(* Logix 5000 project; controller reports 1756-L63 rev 20.15; software revision 20.04; part 8 of 52 *)

        [734].log_data[9].valid := 1, [734].log_data[10].valid := 1, [734].log_data[11].valid := 1, [734].log_data[12].valid := 1, [734].log_data[13].valid := 1, [734].log_data[14].valid := 1, [734].log_data[15].valid := 1, [734].log_data[16].valid := 1, [734].log_data[17].valid := 1, [734].log_data[18].valid := 1, [734].log_data[19].valid := 1, [734].time.Year := 2023, [734].time.Month := 1, [734].time.Day := 15, [734].time.Hour := 7, [734].time.Minute := 59, [734].time.Second := 59, [735].log_data[0].min := 1.0, [735].log_data[0].max := 1.0, [735].log_data[0].total := 900.0, [735].log_data[0].time := 900.0, [735].log_data[0].valid := 1, [735].log_data[1].valid := 1, [735].log_data[2].valid := 1, [735].log_data[3].valid := 1, [735].log_data[4].valid := 1, [735].log_data[5].valid := 1, [735].log_data[6].valid := 1, [735].log_data[7].valid := 1, [735].log_data[8].valid := 1, [735].log_data[9].valid := 1, [735].log_data[10].valid := 1, [735].log_data[11].valid := 1, [735].log_data[12].valid := 1, [735].log_data[13].valid := 1, [735].log_data[14].valid := 1, [735].log_data[15].valid := 1, [735].log_data[16].valid := 1, [735].log_data[17].valid := 1, [735].log_data[18].valid := 1, [735].log_data[19].valid := 1, [735].time.Year := 2023, [735].time.Month := 1, [735].time.Day := 15, [735].time.Hour := 8, [735].time.Minute := 14, [735].time.Second := 59, [736].log_data[0].min := 1.0, [736].log_data[0].max := 1.0, [736].log_data[0].total := 900.0, [736].log_data[0].time := 900.0, [736].log_data[0].minminute := 15, [736].log_data[0].maxminute := 15, [736].log_data[0].valid := 1, [736].log_data[1].valid := 1, [736].log_data[2].valid := 1, [736].log_data[3].valid := 1, [736].log_data[4].valid := 1, [736].log_data[5].valid := 1, [736].log_data[6].valid := 1,
        [736].log_data[7].valid := 1, [736].log_data[8].valid := 1, [736].log_data[9].valid := 1, [736].log_data[10].valid := 1, [736].log_data[11].valid := 1, [736].log_data[12].valid := 1, [736].log_data[13].valid := 1, [736].log_data[14].valid := 1, [736].log_data[15].valid := 1, [736].log_data[16].valid := 1, [736].log_data[17].valid := 1, [736].log_data[18].valid := 1, [736].log_data[19].valid := 1, [736].time.Year := 2023, [736].time.Month := 1, [736].time.Day := 15, [736].time.Hour := 8, [736].time.Minute := 29, [736].time.Second := 59, [737].log_data[0].min := 1.0, [737].log_data[0].max := 1.0, [737].log_data[0].total := 900.0, [737].log_data[0].time := 900.0, [737].log_data[0].minminute := 30, [737].log_data[0].maxminute := 30, [737].log_data[0].valid := 1, [737].log_data[1].valid := 1, [737].log_data[2].valid := 1, [737].log_data[3].valid := 1, [737].log_data[4].valid := 1, [737].log_data[5].valid := 1, [737].log_data[6].valid := 1, [737].log_data[7].valid := 1, [737].log_data[8].valid := 1, [737].log_data[9].valid := 1, [737].log_data[10].valid := 1, [737].log_data[11].valid := 1, [737].log_data[12].valid := 1, [737].log_data[13].valid := 1, [737].log_data[14].valid := 1, [737].log_data[15].valid := 1, [737].log_data[16].valid := 1, [737].log_data[17].valid := 1, [737].log_data[18].valid := 1, [737].log_data[19].valid := 1, [737].time.Year := 2023, [737].time.Month := 1, [737].time.Day := 15, [737].time.Hour := 8, [737].time.Minute := 44, [737].time.Second := 59, [738].log_data[0].min := 1.0, [738].log_data[0].max := 1.0, [738].log_data[0].total := 900.0, [738].log_data[0].time := 900.0, [738].log_data[0].minminute := 45, [738].log_data[0].maxminute := 45, [738].log_data[0].valid := 1, [738].log_data[1].valid := 1, [738].log_data[2].valid := 1,
        [738].log_data[3].valid := 1, [738].log_data[4].valid := 1, [738].log_data[5].valid := 1, [738].log_data[6].valid := 1, [738].log_data[7].valid := 1, [738].log_data[8].valid := 1, [738].log_data[9].valid := 1, [738].log_data[10].valid := 1, [738].log_data[11].valid := 1, [738].log_data[12].valid := 1, [738].log_data[13].valid := 1, [738].log_data[14].valid := 1, [738].log_data[15].valid := 1, [738].log_data[16].valid := 1, [738].log_data[17].valid := 1, [738].log_data[18].valid := 1, [738].log_data[19].valid := 1, [738].time.Year := 2023, [738].time.Month := 1, [738].time.Day := 15, [738].time.Hour := 8, [738].time.Minute := 59, [738].time.Second := 59, [739].log_data[0].min := 1.0, [739].log_data[0].max := 1.0, [739].log_data[0].total := 900.0, [739].log_data[0].time := 900.0, [739].log_data[0].valid := 1, [739].log_data[1].valid := 1, [739].log_data[2].valid := 1, [739].log_data[3].valid := 1, [739].log_data[4].valid := 1, [739].log_data[5].valid := 1, [739].log_data[6].valid := 1, [739].log_data[7].valid := 1, [739].log_data[8].valid := 1, [739].log_data[9].valid := 1, [739].log_data[10].valid := 1, [739].log_data[11].valid := 1, [739].log_data[12].valid := 1, [739].log_data[13].valid := 1, [739].log_data[14].valid := 1, [739].log_data[15].valid := 1, [739].log_data[16].valid := 1, [739].log_data[17].valid := 1, [739].log_data[18].valid := 1, [739].log_data[19].valid := 1, [739].time.Year := 2023, [739].time.Month := 1, [739].time.Day := 15, [739].time.Hour := 9, [739].time.Minute := 14, [739].time.Second := 59, [740].log_data[0].min := 1.0, [740].log_data[0].max := 1.0, [740].log_data[0].total := 900.0, [740].log_data[0].time := 900.0, [740].log_data[0].minminute := 15, [740].log_data[0].maxminute := 15, [740].log_data[0].valid := 1,
        [740].log_data[1].valid := 1, [740].log_data[2].valid := 1, [740].log_data[3].valid := 1, [740].log_data[4].valid := 1, [740].log_data[5].valid := 1, [740].log_data[6].valid := 1, [740].log_data[7].valid := 1, [740].log_data[8].valid := 1, [740].log_data[9].valid := 1, [740].log_data[10].valid := 1, [740].log_data[11].valid := 1, [740].log_data[12].valid := 1, [740].log_data[13].valid := 1, [740].log_data[14].valid := 1, [740].log_data[15].valid := 1, [740].log_data[16].valid := 1, [740].log_data[17].valid := 1, [740].log_data[18].valid := 1, [740].log_data[19].valid := 1, [740].time.Year := 2023, [740].time.Month := 1, [740].time.Day := 15, [740].time.Hour := 9, [740].time.Minute := 29, [740].time.Second := 59, [741].log_data[0].min := 1.0, [741].log_data[0].max := 1.0, [741].log_data[0].total := 900.0, [741].log_data[0].time := 900.0, [741].log_data[0].minminute := 30, [741].log_data[0].maxminute := 30, [741].log_data[0].valid := 1, [741].log_data[1].valid := 1, [741].log_data[2].valid := 1, [741].log_data[3].valid := 1, [741].log_data[4].valid := 1, [741].log_data[5].valid := 1, [741].log_data[6].valid := 1, [741].log_data[7].valid := 1, [741].log_data[8].valid := 1, [741].log_data[9].valid := 1, [741].log_data[10].valid := 1, [741].log_data[11].valid := 1, [741].log_data[12].valid := 1, [741].log_data[13].valid := 1, [741].log_data[14].valid := 1, [741].log_data[15].valid := 1, [741].log_data[16].valid := 1, [741].log_data[17].valid := 1, [741].log_data[18].valid := 1, [741].log_data[19].valid := 1, [741].time.Year := 2023, [741].time.Month := 1, [741].time.Day := 15, [741].time.Hour := 9, [741].time.Minute := 44, [741].time.Second := 59, [742].log_data[0].min := 1.0, [742].log_data[0].max := 1.0, [742].log_data[0].total := 900.0,
        [742].log_data[0].time := 900.0, [742].log_data[0].minminute := 45, [742].log_data[0].maxminute := 45, [742].log_data[0].valid := 1, [742].log_data[1].valid := 1, [742].log_data[2].valid := 1, [742].log_data[3].valid := 1, [742].log_data[4].valid := 1, [742].log_data[5].valid := 1, [742].log_data[6].valid := 1, [742].log_data[7].valid := 1, [742].log_data[8].valid := 1, [742].log_data[9].valid := 1, [742].log_data[10].valid := 1, [742].log_data[11].valid := 1, [742].log_data[12].valid := 1, [742].log_data[13].valid := 1, [742].log_data[14].valid := 1, [742].log_data[15].valid := 1, [742].log_data[16].valid := 1, [742].log_data[17].valid := 1, [742].log_data[18].valid := 1, [742].log_data[19].valid := 1, [742].time.Year := 2023, [742].time.Month := 1, [742].time.Day := 15, [742].time.Hour := 9, [742].time.Minute := 59, [742].time.Second := 59, [743].log_data[0].min := 1.0, [743].log_data[0].max := 1.0, [743].log_data[0].total := 900.0, [743].log_data[0].time := 900.0, [743].log_data[0].valid := 1, [743].log_data[1].valid := 1, [743].log_data[2].valid := 1, [743].log_data[3].valid := 1, [743].log_data[4].valid := 1, [743].log_data[5].valid := 1, [743].log_data[6].valid := 1, [743].log_data[7].valid := 1, [743].log_data[8].valid := 1, [743].log_data[9].valid := 1, [743].log_data[10].valid := 1, [743].log_data[11].valid := 1, [743].log_data[12].valid := 1, [743].log_data[13].valid := 1, [743].log_data[14].valid := 1, [743].log_data[15].valid := 1, [743].log_data[16].valid := 1, [743].log_data[17].valid := 1, [743].log_data[18].valid := 1, [743].log_data[19].valid := 1, [743].time.Year := 2023, [743].time.Month := 1, [743].time.Day := 15, [743].time.Hour := 10, [743].time.Minute := 14, [743].time.Second := 59, [744].log_data[0].min := 1.0,
        [744].log_data[0].max := 1.0, [744].log_data[0].total := 900.0, [744].log_data[0].time := 900.0, [744].log_data[0].minminute := 15, [744].log_data[0].maxminute := 15, [744].log_data[0].valid := 1, [744].log_data[1].valid := 1, [744].log_data[2].valid := 1, [744].log_data[3].valid := 1, [744].log_data[4].valid := 1, [744].log_data[5].valid := 1, [744].log_data[6].valid := 1, [744].log_data[7].valid := 1, [744].log_data[8].valid := 1, [744].log_data[9].valid := 1, [744].log_data[10].valid := 1, [744].log_data[11].valid := 1, [744].log_data[12].valid := 1, [744].log_data[13].valid := 1, [744].log_data[14].valid := 1, [744].log_data[15].valid := 1, [744].log_data[16].valid := 1, [744].log_data[17].valid := 1, [744].log_data[18].valid := 1, [744].log_data[19].valid := 1, [744].time.Year := 2023, [744].time.Month := 1, [744].time.Day := 15, [744].time.Hour := 10, [744].time.Minute := 29, [744].time.Second := 59, [745].log_data[0].min := 1.0, [745].log_data[0].max := 1.0, [745].log_data[0].total := 900.0, [745].log_data[0].time := 900.0, [745].log_data[0].minminute := 30, [745].log_data[0].maxminute := 30, [745].log_data[0].valid := 1, [745].log_data[1].valid := 1, [745].log_data[2].valid := 1, [745].log_data[3].valid := 1, [745].log_data[4].valid := 1, [745].log_data[5].valid := 1, [745].log_data[6].valid := 1, [745].log_data[7].valid := 1, [745].log_data[8].valid := 1, [745].log_data[9].valid := 1, [745].log_data[10].valid := 1, [745].log_data[11].valid := 1, [745].log_data[12].valid := 1, [745].log_data[13].valid := 1, [745].log_data[14].valid := 1, [745].log_data[15].valid := 1, [745].log_data[16].valid := 1, [745].log_data[17].valid := 1, [745].log_data[18].valid := 1, [745].log_data[19].valid := 1, [745].time.Year := 2023, [745].time.Month := 1, [745].time.Day := 15,
        [745].time.Hour := 10, [745].time.Minute := 44, [745].time.Second := 59, [746].log_data[0].min := 1.0, [746].log_data[0].max := 1.0, [746].log_data[0].total := 900.0, [746].log_data[0].time := 900.0, [746].log_data[0].minminute := 45, [746].log_data[0].maxminute := 45, [746].log_data[0].valid := 1, [746].log_data[1].valid := 1, [746].log_data[2].valid := 1, [746].log_data[3].valid := 1, [746].log_data[4].valid := 1, [746].log_data[5].valid := 1, [746].log_data[6].valid := 1, [746].log_data[7].valid := 1, [746].log_data[8].valid := 1, [746].log_data[9].valid := 1, [746].log_data[10].valid := 1, [746].log_data[11].valid := 1, [746].log_data[12].valid := 1, [746].log_data[13].valid := 1, [746].log_data[14].valid := 1, [746].log_data[15].valid := 1, [746].log_data[16].valid := 1, [746].log_data[17].valid := 1, [746].log_data[18].valid := 1, [746].log_data[19].valid := 1, [746].time.Year := 2023, [746].time.Month := 1, [746].time.Day := 15, [746].time.Hour := 10, [746].time.Minute := 59, [746].time.Second := 59, [747].log_data[0].min := 1.0, [747].log_data[0].max := 1.0, [747].log_data[0].total := 899.5, [747].log_data[0].time := 899.5, [747].log_data[0].valid := 1, [747].log_data[1].valid := 1, [747].log_data[2].valid := 1, [747].log_data[3].valid := 1, [747].log_data[4].valid := 1, [747].log_data[5].valid := 1, [747].log_data[6].valid := 1, [747].log_data[7].valid := 1, [747].log_data[8].valid := 1, [747].log_data[9].valid := 1, [747].log_data[10].valid := 1, [747].log_data[11].valid := 1, [747].log_data[12].valid := 1, [747].log_data[13].valid := 1, [747].log_data[14].valid := 1, [747].log_data[15].valid := 1, [747].log_data[16].valid := 1, [747].log_data[17].valid := 1, [747].log_data[18].valid := 1, [747].log_data[19].valid := 1, [747].time.Year := 2023,
        [747].time.Month := 1, [747].time.Day := 15, [747].time.Hour := 11, [747].time.Minute := 14, [747].time.Second := 59, [748].log_data[0].min := 1.0, [748].log_data[0].max := 1.0, [748].log_data[0].total := 900.0, [748].log_data[0].time := 900.0, [748].log_data[0].minminute := 15, [748].log_data[0].maxminute := 15, [748].log_data[0].valid := 1, [748].log_data[1].valid := 1, [748].log_data[2].valid := 1, [748].log_data[3].valid := 1, [748].log_data[4].valid := 1, [748].log_data[5].valid := 1, [748].log_data[6].valid := 1, [748].log_data[7].valid := 1, [748].log_data[8].valid := 1, [748].log_data[9].valid := 1, [748].log_data[10].valid := 1, [748].log_data[11].valid := 1, [748].log_data[12].valid := 1, [748].log_data[13].valid := 1, [748].log_data[14].valid := 1, [748].log_data[15].valid := 1, [748].log_data[16].valid := 1, [748].log_data[17].valid := 1, [748].log_data[18].valid := 1, [748].log_data[19].valid := 1, [748].time.Year := 2023, [748].time.Month := 1, [748].time.Day := 15, [748].time.Hour := 11, [748].time.Minute := 29, [748].time.Second := 59, [749].log_data[0].min := 1.0, [749].log_data[0].max := 1.0, [749].log_data[0].total := 900.0, [749].log_data[0].time := 900.0, [749].log_data[0].minminute := 30, [749].log_data[0].maxminute := 30, [749].log_data[0].valid := 1, [749].log_data[1].valid := 1, [749].log_data[2].valid := 1, [749].log_data[3].valid := 1, [749].log_data[4].valid := 1, [749].log_data[5].valid := 1, [749].log_data[6].valid := 1, [749].log_data[7].valid := 1, [749].log_data[8].valid := 1, [749].log_data[9].valid := 1, [749].log_data[10].valid := 1, [749].log_data[11].valid := 1, [749].log_data[12].valid := 1, [749].log_data[13].valid := 1, [749].log_data[14].valid := 1, [749].log_data[15].valid := 1, [749].log_data[16].valid := 1,
        [749].log_data[17].valid := 1, [749].log_data[18].valid := 1, [749].log_data[19].valid := 1, [749].time.Year := 2023, [749].time.Month := 1, [749].time.Day := 15, [749].time.Hour := 11, [749].time.Minute := 44, [749].time.Second := 59, [750].log_data[0].min := 1.0, [750].log_data[0].max := 1.0, [750].log_data[0].total := 900.0, [750].log_data[0].time := 900.0, [750].log_data[0].minminute := 45, [750].log_data[0].maxminute := 45, [750].log_data[0].valid := 1, [750].log_data[1].valid := 1, [750].log_data[2].valid := 1, [750].log_data[3].valid := 1, [750].log_data[4].valid := 1, [750].log_data[5].valid := 1, [750].log_data[6].valid := 1, [750].log_data[7].valid := 1, [750].log_data[8].valid := 1, [750].log_data[9].valid := 1, [750].log_data[10].valid := 1, [750].log_data[11].valid := 1, [750].log_data[12].valid := 1, [750].log_data[13].valid := 1, [750].log_data[14].valid := 1, [750].log_data[15].valid := 1, [750].log_data[16].valid := 1, [750].log_data[17].valid := 1, [750].log_data[18].valid := 1, [750].log_data[19].valid := 1, [750].time.Year := 2023, [750].time.Month := 1, [750].time.Day := 15, [750].time.Hour := 11, [750].time.Minute := 59, [750].time.Second := 59, [751].log_data[0].min := 1.0, [751].log_data[0].max := 1.0, [751].log_data[0].total := 900.0, [751].log_data[0].time := 900.0, [751].log_data[0].valid := 1, [751].log_data[1].valid := 1, [751].log_data[2].valid := 1, [751].log_data[3].valid := 1, [751].log_data[4].valid := 1, [751].log_data[5].valid := 1, [751].log_data[6].valid := 1, [751].log_data[7].valid := 1, [751].log_data[8].valid := 1, [751].log_data[9].valid := 1, [751].log_data[10].valid := 1, [751].log_data[11].valid := 1, [751].log_data[12].valid := 1, [751].log_data[13].valid := 1, [751].log_data[14].valid := 1,
        [751].log_data[15].valid := 1, [751].log_data[16].valid := 1, [751].log_data[17].valid := 1, [751].log_data[18].valid := 1, [751].log_data[19].valid := 1, [751].time.Year := 2023, [751].time.Month := 1, [751].time.Day := 15, [751].time.Hour := 12, [751].time.Minute := 14, [751].time.Second := 59, [752].log_data[0].min := 1.0, [752].log_data[0].max := 1.0, [752].log_data[0].total := 900.0, [752].log_data[0].time := 900.0, [752].log_data[0].minminute := 15, [752].log_data[0].maxminute := 15, [752].log_data[0].valid := 1, [752].log_data[1].valid := 1, [752].log_data[2].valid := 1, [752].log_data[3].valid := 1, [752].log_data[4].valid := 1, [752].log_data[5].valid := 1, [752].log_data[6].valid := 1, [752].log_data[7].valid := 1, [752].log_data[8].valid := 1, [752].log_data[9].valid := 1, [752].log_data[10].valid := 1, [752].log_data[11].valid := 1, [752].log_data[12].valid := 1, [752].log_data[13].valid := 1, [752].log_data[14].valid := 1, [752].log_data[15].valid := 1, [752].log_data[16].valid := 1, [752].log_data[17].valid := 1, [752].log_data[18].valid := 1, [752].log_data[19].valid := 1, [752].time.Year := 2023, [752].time.Month := 1, [752].time.Day := 15, [752].time.Hour := 12, [752].time.Minute := 29, [752].time.Second := 59, [753].log_data[0].min := 1.0, [753].log_data[0].max := 1.0, [753].log_data[0].total := 900.0, [753].log_data[0].time := 900.0, [753].log_data[0].minminute := 30, [753].log_data[0].maxminute := 30, [753].log_data[0].valid := 1, [753].log_data[1].valid := 1, [753].log_data[2].valid := 1, [753].log_data[3].valid := 1, [753].log_data[4].valid := 1, [753].log_data[5].valid := 1, [753].log_data[6].valid := 1, [753].log_data[7].valid := 1, [753].log_data[8].valid := 1, [753].log_data[9].valid := 1, [753].log_data[10].valid := 1,
        [753].log_data[11].valid := 1, [753].log_data[12].valid := 1, [753].log_data[13].valid := 1, [753].log_data[14].valid := 1, [753].log_data[15].valid := 1, [753].log_data[16].valid := 1, [753].log_data[17].valid := 1, [753].log_data[18].valid := 1, [753].log_data[19].valid := 1, [753].time.Year := 2023, [753].time.Month := 1, [753].time.Day := 15, [753].time.Hour := 12, [753].time.Minute := 44, [753].time.Second := 59, [754].log_data[0].min := 1.0, [754].log_data[0].max := 1.0, [754].log_data[0].total := 900.0, [754].log_data[0].time := 900.0, [754].log_data[0].minminute := 45, [754].log_data[0].maxminute := 45, [754].log_data[0].valid := 1, [754].log_data[1].valid := 1, [754].log_data[2].valid := 1, [754].log_data[3].valid := 1, [754].log_data[4].valid := 1, [754].log_data[5].valid := 1, [754].log_data[6].valid := 1, [754].log_data[7].valid := 1, [754].log_data[8].valid := 1, [754].log_data[9].valid := 1, [754].log_data[10].valid := 1, [754].log_data[11].valid := 1, [754].log_data[12].valid := 1, [754].log_data[13].valid := 1, [754].log_data[14].valid := 1, [754].log_data[15].valid := 1, [754].log_data[16].valid := 1, [754].log_data[17].valid := 1, [754].log_data[18].valid := 1, [754].log_data[19].valid := 1, [754].time.Year := 2023, [754].time.Month := 1, [754].time.Day := 15, [754].time.Hour := 12, [754].time.Minute := 59, [754].time.Second := 59, [755].log_data[0].min := 1.0, [755].log_data[0].max := 1.0, [755].log_data[0].total := 900.0, [755].log_data[0].time := 900.0, [755].log_data[0].valid := 1, [755].log_data[1].valid := 1, [755].log_data[2].valid := 1, [755].log_data[3].valid := 1, [755].log_data[4].valid := 1, [755].log_data[5].valid := 1, [755].log_data[6].valid := 1, [755].log_data[7].valid := 1, [755].log_data[8].valid := 1,
        [755].log_data[9].valid := 1, [755].log_data[10].valid := 1, [755].log_data[11].valid := 1, [755].log_data[12].valid := 1, [755].log_data[13].valid := 1, [755].log_data[14].valid := 1, [755].log_data[15].valid := 1, [755].log_data[16].valid := 1, [755].log_data[17].valid := 1, [755].log_data[18].valid := 1, [755].log_data[19].valid := 1, [755].time.Year := 2023, [755].time.Month := 1, [755].time.Day := 15, [755].time.Hour := 13, [755].time.Minute := 14, [755].time.Second := 59, [756].log_data[0].min := 1.0, [756].log_data[0].max := 1.0, [756].log_data[0].total := 900.0, [756].log_data[0].time := 900.0, [756].log_data[0].minminute := 15, [756].log_data[0].maxminute := 15, [756].log_data[0].valid := 1, [756].log_data[1].valid := 1, [756].log_data[2].valid := 1, [756].log_data[3].valid := 1, [756].log_data[4].valid := 1, [756].log_data[5].valid := 1, [756].log_data[6].valid := 1, [756].log_data[7].valid := 1, [756].log_data[8].valid := 1, [756].log_data[9].valid := 1, [756].log_data[10].valid := 1, [756].log_data[11].valid := 1, [756].log_data[12].valid := 1, [756].log_data[13].valid := 1, [756].log_data[14].valid := 1, [756].log_data[15].valid := 1, [756].log_data[16].valid := 1, [756].log_data[17].valid := 1, [756].log_data[18].valid := 1, [756].log_data[19].valid := 1, [756].time.Year := 2023, [756].time.Month := 1, [756].time.Day := 15, [756].time.Hour := 13, [756].time.Minute := 29, [756].time.Second := 59, [757].log_data[0].min := 1.0, [757].log_data[0].max := 1.0, [757].log_data[0].total := 900.0, [757].log_data[0].time := 900.0, [757].log_data[0].minminute := 30, [757].log_data[0].maxminute := 30, [757].log_data[0].valid := 1, [757].log_data[1].valid := 1, [757].log_data[2].valid := 1, [757].log_data[3].valid := 1, [757].log_data[4].valid := 1,
        [757].log_data[5].valid := 1, [757].log_data[6].valid := 1, [757].log_data[7].valid := 1, [757].log_data[8].valid := 1, [757].log_data[9].valid := 1, [757].log_data[10].valid := 1, [757].log_data[11].valid := 1, [757].log_data[12].valid := 1, [757].log_data[13].valid := 1, [757].log_data[14].valid := 1, [757].log_data[15].valid := 1, [757].log_data[16].valid := 1, [757].log_data[17].valid := 1, [757].log_data[18].valid := 1, [757].log_data[19].valid := 1, [757].time.Year := 2023, [757].time.Month := 1, [757].time.Day := 15, [757].time.Hour := 13, [757].time.Minute := 44, [757].time.Second := 59, [758].log_data[0].min := 1.0, [758].log_data[0].max := 1.0, [758].log_data[0].total := 900.0, [758].log_data[0].time := 900.0, [758].log_data[0].minminute := 45, [758].log_data[0].maxminute := 45, [758].log_data[0].valid := 1, [758].log_data[1].valid := 1, [758].log_data[2].valid := 1, [758].log_data[3].valid := 1, [758].log_data[4].valid := 1, [758].log_data[5].valid := 1, [758].log_data[6].valid := 1, [758].log_data[7].valid := 1, [758].log_data[8].valid := 1, [758].log_data[9].valid := 1, [758].log_data[10].valid := 1, [758].log_data[11].valid := 1, [758].log_data[12].valid := 1, [758].log_data[13].valid := 1, [758].log_data[14].valid := 1, [758].log_data[15].valid := 1, [758].log_data[16].valid := 1, [758].log_data[17].valid := 1, [758].log_data[18].valid := 1, [758].log_data[19].valid := 1, [758].time.Year := 2023, [758].time.Month := 1, [758].time.Day := 15, [758].time.Hour := 13, [758].time.Minute := 59, [758].time.Second := 59, [759].log_data[0].min := 1.0, [759].log_data[0].max := 1.0, [759].log_data[0].total := 900.0, [759].log_data[0].time := 900.0, [759].log_data[0].valid := 1, [759].log_data[1].valid := 1, [759].log_data[2].valid := 1,
        [759].log_data[3].valid := 1, [759].log_data[4].valid := 1, [759].log_data[5].valid := 1, [759].log_data[6].valid := 1, [759].log_data[7].valid := 1, [759].log_data[8].valid := 1, [759].log_data[9].valid := 1, [759].log_data[10].valid := 1, [759].log_data[11].valid := 1, [759].log_data[12].valid := 1, [759].log_data[13].valid := 1, [759].log_data[14].valid := 1, [759].log_data[15].valid := 1, [759].log_data[16].valid := 1, [759].log_data[17].valid := 1, [759].log_data[18].valid := 1, [759].log_data[19].valid := 1, [759].time.Year := 2023, [759].time.Month := 1, [759].time.Day := 15, [759].time.Hour := 14, [759].time.Minute := 14, [759].time.Second := 59, [760].log_data[0].min := 1.0, [760].log_data[0].max := 1.0, [760].log_data[0].total := 900.0, [760].log_data[0].time := 900.0, [760].log_data[0].minminute := 15, [760].log_data[0].maxminute := 15, [760].log_data[0].valid := 1, [760].log_data[1].valid := 1, [760].log_data[2].valid := 1, [760].log_data[3].valid := 1, [760].log_data[4].valid := 1, [760].log_data[5].valid := 1, [760].log_data[6].valid := 1, [760].log_data[7].valid := 1, [760].log_data[8].valid := 1, [760].log_data[9].valid := 1, [760].log_data[10].valid := 1, [760].log_data[11].valid := 1, [760].log_data[12].valid := 1, [760].log_data[13].valid := 1, [760].log_data[14].valid := 1, [760].log_data[15].valid := 1, [760].log_data[16].valid := 1, [760].log_data[17].valid := 1, [760].log_data[18].valid := 1, [760].log_data[19].valid := 1, [760].time.Year := 2023, [760].time.Month := 1, [760].time.Day := 15, [760].time.Hour := 14, [760].time.Minute := 29, [760].time.Second := 59, [761].log_data[0].min := 1.0, [761].log_data[0].max := 1.0, [761].log_data[0].total := 900.0, [761].log_data[0].time := 900.0, [761].log_data[0].minminute := 30,
        [761].log_data[0].maxminute := 30, [761].log_data[0].valid := 1, [761].log_data[1].valid := 1, [761].log_data[2].valid := 1, [761].log_data[3].valid := 1, [761].log_data[4].valid := 1, [761].log_data[5].valid := 1, [761].log_data[6].valid := 1, [761].log_data[7].valid := 1, [761].log_data[8].valid := 1, [761].log_data[9].valid := 1, [761].log_data[10].valid := 1, [761].log_data[11].valid := 1, [761].log_data[12].valid := 1, [761].log_data[13].valid := 1, [761].log_data[14].valid := 1, [761].log_data[15].valid := 1, [761].log_data[16].valid := 1, [761].log_data[17].valid := 1, [761].log_data[18].valid := 1, [761].log_data[19].valid := 1, [761].time.Year := 2023, [761].time.Month := 1, [761].time.Day := 15, [761].time.Hour := 14, [761].time.Minute := 44, [761].time.Second := 59, [762].log_data[0].min := 1.0, [762].log_data[0].max := 1.0, [762].log_data[0].total := 900.0, [762].log_data[0].time := 900.0, [762].log_data[0].minminute := 45, [762].log_data[0].maxminute := 45, [762].log_data[0].valid := 1, [762].log_data[1].valid := 1, [762].log_data[2].valid := 1, [762].log_data[3].valid := 1, [762].log_data[4].valid := 1, [762].log_data[5].valid := 1, [762].log_data[6].valid := 1, [762].log_data[7].valid := 1, [762].log_data[8].valid := 1, [762].log_data[9].valid := 1, [762].log_data[10].valid := 1, [762].log_data[11].valid := 1, [762].log_data[12].valid := 1, [762].log_data[13].valid := 1, [762].log_data[14].valid := 1, [762].log_data[15].valid := 1, [762].log_data[16].valid := 1, [762].log_data[17].valid := 1, [762].log_data[18].valid := 1, [762].log_data[19].valid := 1, [762].time.Year := 2023, [762].time.Month := 1, [762].time.Day := 15, [762].time.Hour := 14, [762].time.Minute := 59, [762].time.Second := 59, [763].log_data[0].min := 1.0,
        [763].log_data[0].max := 1.0, [763].log_data[0].total := 900.0, [763].log_data[0].time := 900.0, [763].log_data[0].valid := 1, [763].log_data[1].valid := 1, [763].log_data[2].valid := 1, [763].log_data[3].valid := 1, [763].log_data[4].valid := 1, [763].log_data[5].valid := 1, [763].log_data[6].valid := 1, [763].log_data[7].valid := 1, [763].log_data[8].valid := 1, [763].log_data[9].valid := 1, [763].log_data[10].valid := 1, [763].log_data[11].valid := 1, [763].log_data[12].valid := 1, [763].log_data[13].valid := 1, [763].log_data[14].valid := 1, [763].log_data[15].valid := 1, [763].log_data[16].valid := 1, [763].log_data[17].valid := 1, [763].log_data[18].valid := 1, [763].log_data[19].valid := 1, [763].time.Year := 2023, [763].time.Month := 1, [763].time.Day := 15, [763].time.Hour := 15, [763].time.Minute := 14, [763].time.Second := 59, [764].log_data[0].min := 1.0, [764].log_data[0].max := 1.0, [764].log_data[0].total := 900.0, [764].log_data[0].time := 900.0, [764].log_data[0].minminute := 15, [764].log_data[0].maxminute := 15, [764].log_data[0].valid := 1, [764].log_data[1].valid := 1, [764].log_data[2].valid := 1, [764].log_data[3].valid := 1, [764].log_data[4].valid := 1, [764].log_data[5].valid := 1, [764].log_data[6].valid := 1, [764].log_data[7].valid := 1, [764].log_data[8].valid := 1, [764].log_data[9].valid := 1, [764].log_data[10].valid := 1, [764].log_data[11].valid := 1, [764].log_data[12].valid := 1, [764].log_data[13].valid := 1, [764].log_data[14].valid := 1, [764].log_data[15].valid := 1, [764].log_data[16].valid := 1, [764].log_data[17].valid := 1, [764].log_data[18].valid := 1, [764].log_data[19].valid := 1, [764].time.Year := 2023, [764].time.Month := 1, [764].time.Day := 15, [764].time.Hour := 15, [764].time.Minute := 29,
        [764].time.Second := 59, [765].log_data[0].min := 1.0, [765].log_data[0].max := 1.0, [765].log_data[0].total := 900.0, [765].log_data[0].time := 900.0, [765].log_data[0].minminute := 30, [765].log_data[0].maxminute := 30, [765].log_data[0].valid := 1, [765].log_data[1].valid := 1, [765].log_data[2].valid := 1, [765].log_data[3].valid := 1, [765].log_data[4].valid := 1, [765].log_data[5].valid := 1, [765].log_data[6].valid := 1, [765].log_data[7].valid := 1, [765].log_data[8].valid := 1, [765].log_data[9].valid := 1, [765].log_data[10].valid := 1, [765].log_data[11].valid := 1, [765].log_data[12].valid := 1, [765].log_data[13].valid := 1, [765].log_data[14].valid := 1, [765].log_data[15].valid := 1, [765].log_data[16].valid := 1, [765].log_data[17].valid := 1, [765].log_data[18].valid := 1, [765].log_data[19].valid := 1, [765].time.Year := 2023, [765].time.Month := 1, [765].time.Day := 15, [765].time.Hour := 15, [765].time.Minute := 44, [765].time.Second := 59, [766].log_data[0].min := 1.0, [766].log_data[0].max := 1.0, [766].log_data[0].total := 900.0, [766].log_data[0].time := 900.0, [766].log_data[0].minminute := 45, [766].log_data[0].maxminute := 45, [766].log_data[0].valid := 1, [766].log_data[1].valid := 1, [766].log_data[2].valid := 1, [766].log_data[3].valid := 1, [766].log_data[4].valid := 1, [766].log_data[5].valid := 1, [766].log_data[6].valid := 1, [766].log_data[7].valid := 1, [766].log_data[8].valid := 1, [766].log_data[9].valid := 1, [766].log_data[10].valid := 1, [766].log_data[11].valid := 1, [766].log_data[12].valid := 1, [766].log_data[13].valid := 1, [766].log_data[14].valid := 1, [766].log_data[15].valid := 1, [766].log_data[16].valid := 1, [766].log_data[17].valid := 1, [766].log_data[18].valid := 1, [766].log_data[19].valid := 1, [766].time.Year := 2023,
        [766].time.Month := 1, [766].time.Day := 15, [766].time.Hour := 15, [766].time.Minute := 59, [766].time.Second := 59, [767].log_data[0].min := 1.0, [767].log_data[0].max := 1.0, [767].log_data[0].total := 900.0, [767].log_data[0].time := 900.0, [767].log_data[0].valid := 1, [767].log_data[1].valid := 1, [767].log_data[2].valid := 1, [767].log_data[3].valid := 1, [767].log_data[4].valid := 1, [767].log_data[5].valid := 1, [767].log_data[6].valid := 1, [767].log_data[7].valid := 1, [767].log_data[8].valid := 1, [767].log_data[9].valid := 1, [767].log_data[10].valid := 1, [767].log_data[11].valid := 1, [767].log_data[12].valid := 1, [767].log_data[13].valid := 1, [767].log_data[14].valid := 1, [767].log_data[15].valid := 1, [767].log_data[16].valid := 1, [767].log_data[17].valid := 1, [767].log_data[18].valid := 1, [767].log_data[19].valid := 1, [767].time.Year := 2023, [767].time.Month := 1, [767].time.Day := 15, [767].time.Hour := 16, [767].time.Minute := 14, [767].time.Second := 59, [768].log_data[0].min := 1.0, [768].log_data[0].max := 1.0, [768].log_data[0].total := 900.0, [768].log_data[0].time := 900.0, [768].log_data[0].minminute := 15, [768].log_data[0].maxminute := 15, [768].log_data[0].valid := 1, [768].log_data[1].valid := 1, [768].log_data[2].valid := 1, [768].log_data[3].valid := 1, [768].log_data[4].valid := 1, [768].log_data[5].valid := 1, [768].log_data[6].valid := 1, [768].log_data[7].valid := 1, [768].log_data[8].valid := 1, [768].log_data[9].valid := 1, [768].log_data[10].valid := 1, [768].log_data[11].valid := 1, [768].log_data[12].valid := 1, [768].log_data[13].valid := 1, [768].log_data[14].valid := 1, [768].log_data[15].valid := 1, [768].log_data[16].valid := 1, [768].log_data[17].valid := 1, [768].log_data[18].valid := 1,
        [768].log_data[19].valid := 1, [768].time.Year := 2023, [768].time.Month := 1, [768].time.Day := 15, [768].time.Hour := 16, [768].time.Minute := 29, [768].time.Second := 59, [769].log_data[0].min := 1.0, [769].log_data[0].max := 1.0, [769].log_data[0].total := 900.0, [769].log_data[0].time := 900.0, [769].log_data[0].minminute := 30, [769].log_data[0].maxminute := 30, [769].log_data[0].valid := 1, [769].log_data[1].valid := 1, [769].log_data[2].valid := 1, [769].log_data[3].valid := 1, [769].log_data[4].valid := 1, [769].log_data[5].valid := 1, [769].log_data[6].valid := 1, [769].log_data[7].valid := 1, [769].log_data[8].valid := 1, [769].log_data[9].valid := 1, [769].log_data[10].valid := 1, [769].log_data[11].valid := 1, [769].log_data[12].valid := 1, [769].log_data[13].valid := 1, [769].log_data[14].valid := 1, [769].log_data[15].valid := 1, [769].log_data[16].valid := 1, [769].log_data[17].valid := 1, [769].log_data[18].valid := 1, [769].log_data[19].valid := 1, [769].time.Year := 2023, [769].time.Month := 1, [769].time.Day := 15, [769].time.Hour := 16, [769].time.Minute := 44, [769].time.Second := 59, [770].log_data[0].min := 1.0, [770].log_data[0].max := 1.0, [770].log_data[0].total := 900.0, [770].log_data[0].time := 900.0, [770].log_data[0].minminute := 45, [770].log_data[0].maxminute := 45, [770].log_data[0].valid := 1, [770].log_data[1].valid := 1, [770].log_data[2].valid := 1, [770].log_data[3].valid := 1, [770].log_data[4].valid := 1, [770].log_data[5].valid := 1, [770].log_data[6].valid := 1, [770].log_data[7].valid := 1, [770].log_data[8].valid := 1, [770].log_data[9].valid := 1, [770].log_data[10].valid := 1, [770].log_data[11].valid := 1, [770].log_data[12].valid := 1, [770].log_data[13].valid := 1, [770].log_data[14].valid := 1,
        [770].log_data[15].valid := 1, [770].log_data[16].valid := 1, [770].log_data[17].valid := 1, [770].log_data[18].valid := 1, [770].log_data[19].valid := 1, [770].time.Year := 2023, [770].time.Month := 1, [770].time.Day := 15, [770].time.Hour := 16, [770].time.Minute := 59, [770].time.Second := 59, [771].log_data[0].min := 1.0, [771].log_data[0].max := 1.0, [771].log_data[0].total := 900.0, [771].log_data[0].time := 900.0, [771].log_data[0].valid := 1, [771].log_data[1].valid := 1, [771].log_data[2].valid := 1, [771].log_data[3].valid := 1, [771].log_data[4].valid := 1, [771].log_data[5].valid := 1, [771].log_data[6].valid := 1, [771].log_data[7].valid := 1, [771].log_data[8].valid := 1, [771].log_data[9].valid := 1, [771].log_data[10].valid := 1, [771].log_data[11].valid := 1, [771].log_data[12].valid := 1, [771].log_data[13].valid := 1, [771].log_data[14].valid := 1, [771].log_data[15].valid := 1, [771].log_data[16].valid := 1, [771].log_data[17].valid := 1, [771].log_data[18].valid := 1, [771].log_data[19].valid := 1, [771].time.Year := 2023, [771].time.Month := 1, [771].time.Day := 15, [771].time.Hour := 17, [771].time.Minute := 14, [771].time.Second := 59, [772].log_data[0].min := 1.0, [772].log_data[0].max := 1.0, [772].log_data[0].total := 900.0, [772].log_data[0].time := 900.0, [772].log_data[0].minminute := 15, [772].log_data[0].maxminute := 15, [772].log_data[0].valid := 1, [772].log_data[1].valid := 1, [772].log_data[2].valid := 1, [772].log_data[3].valid := 1, [772].log_data[4].valid := 1, [772].log_data[5].valid := 1, [772].log_data[6].valid := 1, [772].log_data[7].valid := 1, [772].log_data[8].valid := 1, [772].log_data[9].valid := 1, [772].log_data[10].valid := 1, [772].log_data[11].valid := 1, [772].log_data[12].valid := 1,
        [772].log_data[13].valid := 1, [772].log_data[14].valid := 1, [772].log_data[15].valid := 1, [772].log_data[16].valid := 1, [772].log_data[17].valid := 1, [772].log_data[18].valid := 1, [772].log_data[19].valid := 1, [772].time.Year := 2023, [772].time.Month := 1, [772].time.Day := 15, [772].time.Hour := 17, [772].time.Minute := 29, [772].time.Second := 59, [773].log_data[0].min := 1.0, [773].log_data[0].max := 1.0, [773].log_data[0].total := 900.0, [773].log_data[0].time := 900.0, [773].log_data[0].minminute := 30, [773].log_data[0].maxminute := 30, [773].log_data[0].valid := 1, [773].log_data[1].valid := 1, [773].log_data[2].valid := 1, [773].log_data[3].valid := 1, [773].log_data[4].valid := 1, [773].log_data[5].valid := 1, [773].log_data[6].valid := 1, [773].log_data[7].valid := 1, [773].log_data[8].valid := 1, [773].log_data[9].valid := 1, [773].log_data[10].valid := 1, [773].log_data[11].valid := 1, [773].log_data[12].valid := 1, [773].log_data[13].valid := 1, [773].log_data[14].valid := 1, [773].log_data[15].valid := 1, [773].log_data[16].valid := 1, [773].log_data[17].valid := 1, [773].log_data[18].valid := 1, [773].log_data[19].valid := 1, [773].time.Year := 2023, [773].time.Month := 1, [773].time.Day := 15, [773].time.Hour := 17, [773].time.Minute := 44, [773].time.Second := 59, [774].log_data[0].min := 1.0, [774].log_data[0].max := 1.0, [774].log_data[0].total := 900.0, [774].log_data[0].time := 900.0, [774].log_data[0].minminute := 45, [774].log_data[0].maxminute := 45, [774].log_data[0].valid := 1, [774].log_data[1].valid := 1, [774].log_data[2].valid := 1, [774].log_data[3].valid := 1, [774].log_data[4].valid := 1, [774].log_data[5].valid := 1, [774].log_data[6].valid := 1, [774].log_data[7].valid := 1, [774].log_data[8].valid := 1,
        [774].log_data[9].valid := 1, [774].log_data[10].valid := 1, [774].log_data[11].valid := 1, [774].log_data[12].valid := 1, [774].log_data[13].valid := 1, [774].log_data[14].valid := 1, [774].log_data[15].valid := 1, [774].log_data[16].valid := 1, [774].log_data[17].valid := 1, [774].log_data[18].valid := 1, [774].log_data[19].valid := 1, [774].time.Year := 2023, [774].time.Month := 1, [774].time.Day := 15, [774].time.Hour := 17, [774].time.Minute := 59, [774].time.Second := 59, [775].log_data[0].min := 1.0, [775].log_data[0].max := 1.0, [775].log_data[0].total := 900.0, [775].log_data[0].time := 900.0, [775].log_data[0].valid := 1, [775].log_data[1].valid := 1, [775].log_data[2].valid := 1, [775].log_data[3].valid := 1, [775].log_data[4].valid := 1, [775].log_data[5].valid := 1, [775].log_data[6].valid := 1, [775].log_data[7].valid := 1, [775].log_data[8].valid := 1, [775].log_data[9].valid := 1, [775].log_data[10].valid := 1, [775].log_data[11].valid := 1, [775].log_data[12].valid := 1, [775].log_data[13].valid := 1, [775].log_data[14].valid := 1, [775].log_data[15].valid := 1, [775].log_data[16].valid := 1, [775].log_data[17].valid := 1, [775].log_data[18].valid := 1, [775].log_data[19].valid := 1, [775].time.Year := 2023, [775].time.Month := 1, [775].time.Day := 15, [775].time.Hour := 18, [775].time.Minute := 14, [775].time.Second := 59, [776].log_data[0].min := 1.0, [776].log_data[0].max := 1.0, [776].log_data[0].total := 900.0, [776].log_data[0].time := 900.0, [776].log_data[0].minminute := 15, [776].log_data[0].maxminute := 15, [776].log_data[0].valid := 1, [776].log_data[1].valid := 1, [776].log_data[2].valid := 1, [776].log_data[3].valid := 1, [776].log_data[4].valid := 1, [776].log_data[5].valid := 1, [776].log_data[6].valid := 1,
        [776].log_data[7].valid := 1, [776].log_data[8].valid := 1, [776].log_data[9].valid := 1, [776].log_data[10].valid := 1, [776].log_data[11].valid := 1, [776].log_data[12].valid := 1, [776].log_data[13].valid := 1, [776].log_data[14].valid := 1, [776].log_data[15].valid := 1, [776].log_data[16].valid := 1, [776].log_data[17].valid := 1, [776].log_data[18].valid := 1, [776].log_data[19].valid := 1, [776].time.Year := 2023, [776].time.Month := 1, [776].time.Day := 15, [776].time.Hour := 18, [776].time.Minute := 29, [776].time.Second := 59, [777].log_data[0].min := 1.0, [777].log_data[0].max := 1.0, [777].log_data[0].total := 900.0, [777].log_data[0].time := 900.0, [777].log_data[0].minminute := 30, [777].log_data[0].maxminute := 30, [777].log_data[0].valid := 1, [777].log_data[1].valid := 1, [777].log_data[2].valid := 1, [777].log_data[3].valid := 1, [777].log_data[4].valid := 1, [777].log_data[5].valid := 1, [777].log_data[6].valid := 1, [777].log_data[7].valid := 1, [777].log_data[8].valid := 1, [777].log_data[9].valid := 1, [777].log_data[10].valid := 1, [777].log_data[11].valid := 1, [777].log_data[12].valid := 1, [777].log_data[13].valid := 1, [777].log_data[14].valid := 1, [777].log_data[15].valid := 1, [777].log_data[16].valid := 1, [777].log_data[17].valid := 1, [777].log_data[18].valid := 1, [777].log_data[19].valid := 1, [777].time.Year := 2023, [777].time.Month := 1, [777].time.Day := 15, [777].time.Hour := 18, [777].time.Minute := 44, [777].time.Second := 59, [778].log_data[0].min := 1.0, [778].log_data[0].max := 1.0, [778].log_data[0].total := 900.0, [778].log_data[0].time := 900.0, [778].log_data[0].minminute := 45, [778].log_data[0].maxminute := 45, [778].log_data[0].valid := 1, [778].log_data[1].valid := 1, [778].log_data[2].valid := 1,
        [778].log_data[3].valid := 1, [778].log_data[4].valid := 1, [778].log_data[5].valid := 1, [778].log_data[6].valid := 1, [778].log_data[7].valid := 1, [778].log_data[8].valid := 1, [778].log_data[9].valid := 1, [778].log_data[10].valid := 1, [778].log_data[11].valid := 1, [778].log_data[12].valid := 1, [778].log_data[13].valid := 1, [778].log_data[14].valid := 1, [778].log_data[15].valid := 1, [778].log_data[16].valid := 1, [778].log_data[17].valid := 1, [778].log_data[18].valid := 1, [778].log_data[19].valid := 1, [778].time.Year := 2023, [778].time.Month := 1, [778].time.Day := 15, [778].time.Hour := 18, [778].time.Minute := 59, [778].time.Second := 59, [779].log_data[0].min := 1.0, [779].log_data[0].max := 1.0, [779].log_data[0].total := 900.0, [779].log_data[0].time := 900.0, [779].log_data[0].valid := 1, [779].log_data[1].valid := 1, [779].log_data[2].valid := 1, [779].log_data[3].valid := 1, [779].log_data[4].valid := 1, [779].log_data[5].valid := 1, [779].log_data[6].valid := 1, [779].log_data[7].valid := 1, [779].log_data[8].valid := 1, [779].log_data[9].valid := 1, [779].log_data[10].valid := 1, [779].log_data[11].valid := 1, [779].log_data[12].valid := 1, [779].log_data[13].valid := 1, [779].log_data[14].valid := 1, [779].log_data[15].valid := 1, [779].log_data[16].valid := 1, [779].log_data[17].valid := 1, [779].log_data[18].valid := 1, [779].log_data[19].valid := 1, [779].time.Year := 2023, [779].time.Month := 1, [779].time.Day := 15, [779].time.Hour := 19, [779].time.Minute := 14, [779].time.Second := 59, [780].log_data[0].min := 1.0, [780].log_data[0].max := 1.0, [780].log_data[0].total := 900.0, [780].log_data[0].time := 900.0, [780].log_data[0].minminute := 15, [780].log_data[0].maxminute := 15, [780].log_data[0].valid := 1,
        [780].log_data[1].valid := 1, [780].log_data[2].valid := 1, [780].log_data[3].valid := 1, [780].log_data[4].valid := 1, [780].log_data[5].valid := 1, [780].log_data[6].valid := 1, [780].log_data[7].valid := 1, [780].log_data[8].valid := 1, [780].log_data[9].valid := 1, [780].log_data[10].valid := 1, [780].log_data[11].valid := 1, [780].log_data[12].valid := 1, [780].log_data[13].valid := 1, [780].log_data[14].valid := 1, [780].log_data[15].valid := 1, [780].log_data[16].valid := 1, [780].log_data[17].valid := 1, [780].log_data[18].valid := 1, [780].log_data[19].valid := 1, [780].time.Year := 2023, [780].time.Month := 1, [780].time.Day := 15, [780].time.Hour := 19, [780].time.Minute := 29, [780].time.Second := 59, [781].log_data[0].min := 1.0, [781].log_data[0].max := 1.0, [781].log_data[0].total := 900.0, [781].log_data[0].time := 900.0, [781].log_data[0].minminute := 30, [781].log_data[0].maxminute := 30, [781].log_data[0].valid := 1, [781].log_data[1].valid := 1, [781].log_data[2].valid := 1, [781].log_data[3].valid := 1, [781].log_data[4].valid := 1, [781].log_data[5].valid := 1, [781].log_data[6].valid := 1, [781].log_data[7].valid := 1, [781].log_data[8].valid := 1, [781].log_data[9].valid := 1, [781].log_data[10].valid := 1, [781].log_data[11].valid := 1, [781].log_data[12].valid := 1, [781].log_data[13].valid := 1, [781].log_data[14].valid := 1, [781].log_data[15].valid := 1, [781].log_data[16].valid := 1, [781].log_data[17].valid := 1, [781].log_data[18].valid := 1, [781].log_data[19].valid := 1, [781].time.Year := 2023, [781].time.Month := 1, [781].time.Day := 15, [781].time.Hour := 19, [781].time.Minute := 44, [781].time.Second := 59, [782].log_data[0].min := 1.0, [782].log_data[0].max := 1.0, [782].log_data[0].total := 900.0,
        [782].log_data[0].time := 900.0, [782].log_data[0].minminute := 45, [782].log_data[0].maxminute := 45, [782].log_data[0].valid := 1, [782].log_data[1].valid := 1, [782].log_data[2].valid := 1, [782].log_data[3].valid := 1, [782].log_data[4].valid := 1, [782].log_data[5].valid := 1, [782].log_data[6].valid := 1, [782].log_data[7].valid := 1, [782].log_data[8].valid := 1, [782].log_data[9].valid := 1, [782].log_data[10].valid := 1, [782].log_data[11].valid := 1, [782].log_data[12].valid := 1, [782].log_data[13].valid := 1, [782].log_data[14].valid := 1, [782].log_data[15].valid := 1, [782].log_data[16].valid := 1, [782].log_data[17].valid := 1, [782].log_data[18].valid := 1, [782].log_data[19].valid := 1, [782].time.Year := 2023, [782].time.Month := 1, [782].time.Day := 15, [782].time.Hour := 19, [782].time.Minute := 59, [782].time.Second := 59, [783].log_data[0].min := 1.0, [783].log_data[0].max := 1.0, [783].log_data[0].total := 900.0, [783].log_data[0].time := 900.0, [783].log_data[0].valid := 1, [783].log_data[1].valid := 1, [783].log_data[2].valid := 1, [783].log_data[3].valid := 1, [783].log_data[4].valid := 1, [783].log_data[5].valid := 1, [783].log_data[6].valid := 1, [783].log_data[7].valid := 1, [783].log_data[8].valid := 1, [783].log_data[9].valid := 1, [783].log_data[10].valid := 1, [783].log_data[11].valid := 1, [783].log_data[12].valid := 1, [783].log_data[13].valid := 1, [783].log_data[14].valid := 1, [783].log_data[15].valid := 1, [783].log_data[16].valid := 1, [783].log_data[17].valid := 1, [783].log_data[18].valid := 1, [783].log_data[19].valid := 1, [783].time.Year := 2023, [783].time.Month := 1, [783].time.Day := 15, [783].time.Hour := 20, [783].time.Minute := 14, [783].time.Second := 59, [784].log_data[0].min := 1.0,
        [784].log_data[0].max := 1.0, [784].log_data[0].total := 900.0, [784].log_data[0].time := 900.0, [784].log_data[0].minminute := 15, [784].log_data[0].maxminute := 15, [784].log_data[0].valid := 1, [784].log_data[1].valid := 1, [784].log_data[2].valid := 1, [784].log_data[3].valid := 1, [784].log_data[4].valid := 1, [784].log_data[5].valid := 1, [784].log_data[6].valid := 1, [784].log_data[7].valid := 1, [784].log_data[8].valid := 1, [784].log_data[9].valid := 1, [784].log_data[10].valid := 1, [784].log_data[11].valid := 1, [784].log_data[12].valid := 1, [784].log_data[13].valid := 1, [784].log_data[14].valid := 1, [784].log_data[15].valid := 1, [784].log_data[16].valid := 1, [784].log_data[17].valid := 1, [784].log_data[18].valid := 1, [784].log_data[19].valid := 1, [784].time.Year := 2023, [784].time.Month := 1, [784].time.Day := 15, [784].time.Hour := 20, [784].time.Minute := 29, [784].time.Second := 59, [785].log_data[0].min := 1.0, [785].log_data[0].max := 1.0, [785].log_data[0].total := 900.0, [785].log_data[0].time := 900.0, [785].log_data[0].minminute := 30, [785].log_data[0].maxminute := 30, [785].log_data[0].valid := 1, [785].log_data[1].valid := 1, [785].log_data[2].valid := 1, [785].log_data[3].valid := 1, [785].log_data[4].valid := 1, [785].log_data[5].valid := 1, [785].log_data[6].valid := 1, [785].log_data[7].valid := 1, [785].log_data[8].valid := 1, [785].log_data[9].valid := 1, [785].log_data[10].valid := 1, [785].log_data[11].valid := 1, [785].log_data[12].valid := 1, [785].log_data[13].valid := 1, [785].log_data[14].valid := 1, [785].log_data[15].valid := 1, [785].log_data[16].valid := 1, [785].log_data[17].valid := 1, [785].log_data[18].valid := 1, [785].log_data[19].valid := 1, [785].time.Year := 2023, [785].time.Month := 1, [785].time.Day := 15,
        [785].time.Hour := 20, [785].time.Minute := 44, [785].time.Second := 59, [786].log_data[0].min := 1.0, [786].log_data[0].max := 1.0, [786].log_data[0].total := 900.0, [786].log_data[0].time := 900.0, [786].log_data[0].minminute := 45, [786].log_data[0].maxminute := 45, [786].log_data[0].valid := 1, [786].log_data[1].valid := 1, [786].log_data[2].valid := 1, [786].log_data[3].valid := 1, [786].log_data[4].valid := 1, [786].log_data[5].valid := 1, [786].log_data[6].valid := 1, [786].log_data[7].valid := 1, [786].log_data[8].valid := 1, [786].log_data[9].valid := 1, [786].log_data[10].valid := 1, [786].log_data[11].valid := 1, [786].log_data[12].valid := 1, [786].log_data[13].valid := 1, [786].log_data[14].valid := 1, [786].log_data[15].valid := 1, [786].log_data[16].valid := 1, [786].log_data[17].valid := 1, [786].log_data[18].valid := 1, [786].log_data[19].valid := 1, [786].time.Year := 2023, [786].time.Month := 1, [786].time.Day := 15, [786].time.Hour := 20, [786].time.Minute := 59, [786].time.Second := 59, [787].log_data[0].min := 1.0, [787].log_data[0].max := 1.0, [787].log_data[0].total := 900.0, [787].log_data[0].time := 900.0, [787].log_data[0].valid := 1, [787].log_data[1].valid := 1, [787].log_data[2].valid := 1, [787].log_data[3].valid := 1, [787].log_data[4].valid := 1, [787].log_data[5].valid := 1, [787].log_data[6].valid := 1, [787].log_data[7].valid := 1, [787].log_data[8].valid := 1, [787].log_data[9].valid := 1, [787].log_data[10].valid := 1, [787].log_data[11].valid := 1, [787].log_data[12].valid := 1, [787].log_data[13].valid := 1, [787].log_data[14].valid := 1, [787].log_data[15].valid := 1, [787].log_data[16].valid := 1, [787].log_data[17].valid := 1, [787].log_data[18].valid := 1, [787].log_data[19].valid := 1, [787].time.Year := 2023,
        [787].time.Month := 1, [787].time.Day := 15, [787].time.Hour := 21, [787].time.Minute := 14, [787].time.Second := 59, [788].log_data[0].min := 1.0, [788].log_data[0].max := 1.0, [788].log_data[0].total := 900.0, [788].log_data[0].time := 900.0, [788].log_data[0].minminute := 15, [788].log_data[0].maxminute := 15, [788].log_data[0].valid := 1, [788].log_data[1].valid := 1, [788].log_data[2].valid := 1, [788].log_data[3].valid := 1, [788].log_data[4].valid := 1, [788].log_data[5].valid := 1, [788].log_data[6].valid := 1, [788].log_data[7].valid := 1, [788].log_data[8].valid := 1, [788].log_data[9].valid := 1, [788].log_data[10].valid := 1, [788].log_data[11].valid := 1, [788].log_data[12].valid := 1, [788].log_data[13].valid := 1, [788].log_data[14].valid := 1, [788].log_data[15].valid := 1, [788].log_data[16].valid := 1, [788].log_data[17].valid := 1, [788].log_data[18].valid := 1, [788].log_data[19].valid := 1, [788].time.Year := 2023, [788].time.Month := 1, [788].time.Day := 15, [788].time.Hour := 21, [788].time.Minute := 29, [788].time.Second := 59, [789].log_data[0].min := 1.0, [789].log_data[0].max := 1.0, [789].log_data[0].total := 900.0, [789].log_data[0].time := 900.0, [789].log_data[0].minminute := 30, [789].log_data[0].maxminute := 30, [789].log_data[0].valid := 1, [789].log_data[1].valid := 1, [789].log_data[2].valid := 1, [789].log_data[3].valid := 1, [789].log_data[4].valid := 1, [789].log_data[5].valid := 1, [789].log_data[6].valid := 1, [789].log_data[7].valid := 1, [789].log_data[8].valid := 1, [789].log_data[9].valid := 1, [789].log_data[10].valid := 1, [789].log_data[11].valid := 1, [789].log_data[12].valid := 1, [789].log_data[13].valid := 1, [789].log_data[14].valid := 1, [789].log_data[15].valid := 1, [789].log_data[16].valid := 1,
        [789].log_data[17].valid := 1, [789].log_data[18].valid := 1, [789].log_data[19].valid := 1, [789].time.Year := 2023, [789].time.Month := 1, [789].time.Day := 15, [789].time.Hour := 21, [789].time.Minute := 44, [789].time.Second := 59, [790].log_data[0].min := 1.0, [790].log_data[0].max := 1.0, [790].log_data[0].total := 900.0, [790].log_data[0].time := 900.0, [790].log_data[0].minminute := 45, [790].log_data[0].maxminute := 45, [790].log_data[0].valid := 1, [790].log_data[1].valid := 1, [790].log_data[2].valid := 1, [790].log_data[3].valid := 1, [790].log_data[4].valid := 1, [790].log_data[5].valid := 1, [790].log_data[6].valid := 1, [790].log_data[7].valid := 1, [790].log_data[8].valid := 1, [790].log_data[9].valid := 1, [790].log_data[10].valid := 1, [790].log_data[11].valid := 1, [790].log_data[12].valid := 1, [790].log_data[13].valid := 1, [790].log_data[14].valid := 1, [790].log_data[15].valid := 1, [790].log_data[16].valid := 1, [790].log_data[17].valid := 1, [790].log_data[18].valid := 1, [790].log_data[19].valid := 1, [790].time.Year := 2023, [790].time.Month := 1, [790].time.Day := 15, [790].time.Hour := 21, [790].time.Minute := 59, [790].time.Second := 59, [791].log_data[0].min := 1.0, [791].log_data[0].max := 1.0, [791].log_data[0].total := 899.5, [791].log_data[0].time := 899.5, [791].log_data[0].valid := 1, [791].log_data[1].valid := 1, [791].log_data[2].valid := 1, [791].log_data[3].valid := 1, [791].log_data[4].valid := 1, [791].log_data[5].valid := 1, [791].log_data[6].valid := 1, [791].log_data[7].valid := 1, [791].log_data[8].valid := 1, [791].log_data[9].valid := 1, [791].log_data[10].valid := 1, [791].log_data[11].valid := 1, [791].log_data[12].valid := 1, [791].log_data[13].valid := 1, [791].log_data[14].valid := 1,
        [791].log_data[15].valid := 1, [791].log_data[16].valid := 1, [791].log_data[17].valid := 1, [791].log_data[18].valid := 1, [791].log_data[19].valid := 1, [791].time.Year := 2023, [791].time.Month := 1, [791].time.Day := 15, [791].time.Hour := 22, [791].time.Minute := 14, [791].time.Second := 59, [792].log_data[0].min := 1.0, [792].log_data[0].max := 1.0, [792].log_data[0].total := 900.0, [792].log_data[0].time := 900.0, [792].log_data[0].minminute := 15, [792].log_data[0].maxminute := 15, [792].log_data[0].valid := 1, [792].log_data[1].valid := 1, [792].log_data[2].valid := 1, [792].log_data[3].valid := 1, [792].log_data[4].valid := 1, [792].log_data[5].valid := 1, [792].log_data[6].valid := 1, [792].log_data[7].valid := 1, [792].log_data[8].valid := 1, [792].log_data[9].valid := 1, [792].log_data[10].valid := 1, [792].log_data[11].valid := 1, [792].log_data[12].valid := 1, [792].log_data[13].valid := 1, [792].log_data[14].valid := 1, [792].log_data[15].valid := 1, [792].log_data[16].valid := 1, [792].log_data[17].valid := 1, [792].log_data[18].valid := 1, [792].log_data[19].valid := 1, [792].time.Year := 2023, [792].time.Month := 1, [792].time.Day := 15, [792].time.Hour := 22, [792].time.Minute := 29, [792].time.Second := 59, [793].log_data[0].min := 1.0, [793].log_data[0].max := 1.0, [793].log_data[0].total := 900.0, [793].log_data[0].time := 900.0, [793].log_data[0].minminute := 30, [793].log_data[0].maxminute := 30, [793].log_data[0].valid := 1, [793].log_data[1].valid := 1, [793].log_data[2].valid := 1, [793].log_data[3].valid := 1, [793].log_data[4].valid := 1, [793].log_data[5].valid := 1, [793].log_data[6].valid := 1, [793].log_data[7].valid := 1, [793].log_data[8].valid := 1, [793].log_data[9].valid := 1, [793].log_data[10].valid := 1,
        [793].log_data[11].valid := 1, [793].log_data[12].valid := 1, [793].log_data[13].valid := 1, [793].log_data[14].valid := 1, [793].log_data[15].valid := 1, [793].log_data[16].valid := 1, [793].log_data[17].valid := 1, [793].log_data[18].valid := 1, [793].log_data[19].valid := 1, [793].time.Year := 2023, [793].time.Month := 1, [793].time.Day := 15, [793].time.Hour := 22, [793].time.Minute := 44, [793].time.Second := 59, [794].log_data[0].min := 1.0, [794].log_data[0].max := 1.0, [794].log_data[0].total := 900.0, [794].log_data[0].time := 900.0, [794].log_data[0].minminute := 45, [794].log_data[0].maxminute := 45, [794].log_data[0].valid := 1, [794].log_data[1].valid := 1, [794].log_data[2].valid := 1, [794].log_data[3].valid := 1, [794].log_data[4].valid := 1, [794].log_data[5].valid := 1, [794].log_data[6].valid := 1, [794].log_data[7].valid := 1, [794].log_data[8].valid := 1, [794].log_data[9].valid := 1, [794].log_data[10].valid := 1, [794].log_data[11].valid := 1, [794].log_data[12].valid := 1, [794].log_data[13].valid := 1, [794].log_data[14].valid := 1, [794].log_data[15].valid := 1, [794].log_data[16].valid := 1, [794].log_data[17].valid := 1, [794].log_data[18].valid := 1, [794].log_data[19].valid := 1, [794].time.Year := 2023, [794].time.Month := 1, [794].time.Day := 15, [794].time.Hour := 22, [794].time.Minute := 59, [794].time.Second := 59, [795].log_data[0].min := 1.0, [795].log_data[0].max := 1.0, [795].log_data[0].total := 900.0, [795].log_data[0].time := 900.0, [795].log_data[0].valid := 1, [795].log_data[1].valid := 1, [795].log_data[2].valid := 1, [795].log_data[3].valid := 1, [795].log_data[4].valid := 1, [795].log_data[5].valid := 1, [795].log_data[6].valid := 1, [795].log_data[7].valid := 1, [795].log_data[8].valid := 1,
        [795].log_data[9].valid := 1, [795].log_data[10].valid := 1, [795].log_data[11].valid := 1, [795].log_data[12].valid := 1, [795].log_data[13].valid := 1, [795].log_data[14].valid := 1, [795].log_data[15].valid := 1, [795].log_data[16].valid := 1, [795].log_data[17].valid := 1, [795].log_data[18].valid := 1, [795].log_data[19].valid := 1, [795].time.Year := 2023, [795].time.Month := 1, [795].time.Day := 15, [795].time.Hour := 23, [795].time.Minute := 14, [795].time.Second := 59, [796].log_data[0].min := 1.0, [796].log_data[0].max := 1.0, [796].log_data[0].total := 900.0, [796].log_data[0].time := 900.0, [796].log_data[0].minminute := 15, [796].log_data[0].maxminute := 15, [796].log_data[0].valid := 1, [796].log_data[1].valid := 1, [796].log_data[2].valid := 1, [796].log_data[3].valid := 1, [796].log_data[4].valid := 1, [796].log_data[5].valid := 1, [796].log_data[6].valid := 1, [796].log_data[7].valid := 1, [796].log_data[8].valid := 1, [796].log_data[9].valid := 1, [796].log_data[10].valid := 1, [796].log_data[11].valid := 1, [796].log_data[12].valid := 1, [796].log_data[13].valid := 1, [796].log_data[14].valid := 1, [796].log_data[15].valid := 1, [796].log_data[16].valid := 1, [796].log_data[17].valid := 1, [796].log_data[18].valid := 1, [796].log_data[19].valid := 1, [796].time.Year := 2023, [796].time.Month := 1, [796].time.Day := 15, [796].time.Hour := 23, [796].time.Minute := 29, [796].time.Second := 59, [797].log_data[0].min := 1.0, [797].log_data[0].max := 1.0, [797].log_data[0].total := 900.0, [797].log_data[0].time := 900.0, [797].log_data[0].minminute := 30, [797].log_data[0].maxminute := 30, [797].log_data[0].valid := 1, [797].log_data[1].valid := 1, [797].log_data[2].valid := 1, [797].log_data[3].valid := 1, [797].log_data[4].valid := 1,
        [797].log_data[5].valid := 1, [797].log_data[6].valid := 1, [797].log_data[7].valid := 1, [797].log_data[8].valid := 1, [797].log_data[9].valid := 1, [797].log_data[10].valid := 1, [797].log_data[11].valid := 1, [797].log_data[12].valid := 1, [797].log_data[13].valid := 1, [797].log_data[14].valid := 1, [797].log_data[15].valid := 1, [797].log_data[16].valid := 1, [797].log_data[17].valid := 1, [797].log_data[18].valid := 1, [797].log_data[19].valid := 1, [797].time.Year := 2023, [797].time.Month := 1, [797].time.Day := 15, [797].time.Hour := 23, [797].time.Minute := 44, [797].time.Second := 59, [798].log_data[0].min := 1.0, [798].log_data[0].max := 1.0, [798].log_data[0].total := 900.0, [798].log_data[0].time := 900.0, [798].log_data[0].minminute := 45, [798].log_data[0].maxminute := 45, [798].log_data[0].valid := 1, [798].log_data[1].valid := 1, [798].log_data[2].valid := 1, [798].log_data[3].valid := 1, [798].log_data[4].valid := 1, [798].log_data[5].valid := 1, [798].log_data[6].valid := 1, [798].log_data[7].valid := 1, [798].log_data[8].valid := 1, [798].log_data[9].valid := 1, [798].log_data[10].valid := 1, [798].log_data[11].valid := 1, [798].log_data[12].valid := 1, [798].log_data[13].valid := 1, [798].log_data[14].valid := 1, [798].log_data[15].valid := 1, [798].log_data[16].valid := 1, [798].log_data[17].valid := 1, [798].log_data[18].valid := 1, [798].log_data[19].valid := 1, [798].time.Year := 2023, [798].time.Month := 1, [798].time.Day := 15, [798].time.Hour := 23, [798].time.Minute := 59, [798].time.Second := 59, [799].log_data[0].min := 1.0, [799].log_data[0].max := 1.0, [799].log_data[0].total := 900.0, [799].log_data[0].time := 900.0, [799].log_data[0].valid := 1, [799].log_data[1].valid := 1, [799].log_data[2].valid := 1,
        [799].log_data[3].valid := 1, [799].log_data[4].valid := 1, [799].log_data[5].valid := 1, [799].log_data[6].valid := 1, [799].log_data[7].valid := 1, [799].log_data[8].valid := 1, [799].log_data[9].valid := 1, [799].log_data[10].valid := 1, [799].log_data[11].valid := 1, [799].log_data[12].valid := 1, [799].log_data[13].valid := 1, [799].log_data[14].valid := 1, [799].log_data[15].valid := 1, [799].log_data[16].valid := 1, [799].log_data[17].valid := 1, [799].log_data[18].valid := 1, [799].log_data[19].valid := 1, [799].time.Year := 2023, [799].time.Month := 1, [799].time.Day := 16, [799].time.Minute := 14, [799].time.Second := 59);
   report15_row_qty : DINT := 800;
   report5_data : LogRecord5[2400] := ([0].log_data[0].min := 1.0, [0].log_data[0].max := 1.0, [0].log_data[0].total := 300.0, [0].log_data[0].time := 300.0, [0].log_data[0].minminute := 20, [0].log_data[0].maxminute := 20, [0].log_data[0].valid := 1, [0].log_data[1].valid := 1, [0].log_data[2].valid := 1, [0].log_data[3].valid := 1, [0].log_data[4].valid := 1, [0].log_data[5].valid := 1, [0].log_data[6].valid := 1, [0].log_data[7].valid := 1, [0].log_data[8].valid := 1, [0].log_data[9].valid := 1, [0].log_data[10].valid := 1, [0].log_data[11].valid := 1, [0].log_data[12].valid := 1, [0].log_data[13].valid := 1, [0].log_data[14].valid := 1, [0].log_data[15].valid := 1, [0].log_data[16].valid := 1, [0].log_data[17].valid := 1, [0].log_data[18].valid := 1, [0].log_data[19].valid := 1, [0].time.Year := 2023, [0].time.Month := 1, [0].time.Day := 18, [0].time.Minute := 24, [0].time.Second := 59, [1].log_data[0].min := 1.0, [1].log_data[0].max := 1.0, [1].log_data[0].total := 300.0, [1].log_data[0].time := 300.0, [1].log_data[0].minminute := 25, [1].log_data[0].maxminute := 25, [1].log_data[0].valid := 1, [1].log_data[1].valid := 1, [1].log_data[2].valid := 1, [1].log_data[3].valid := 1, [1].log_data[4].valid := 1, [1].log_data[5].valid := 1, [1].log_data[6].valid := 1, [1].log_data[7].valid := 1, [1].log_data[8].valid := 1, [1].log_data[9].valid := 1, [1].log_data[10].valid := 1, [1].log_data[11].valid := 1, [1].log_data[12].valid := 1, [1].log_data[13].valid := 1, [1].log_data[14].valid := 1, [1].log_data[15].valid := 1, [1].log_data[16].valid := 1, [1].log_data[17].valid := 1, [1].log_data[18].valid := 1, [1].log_data[19].valid := 1, [1].time.Year := 2023, [1].time.Month := 1, [1].time.Day := 18,
        [1].time.Minute := 29, [1].time.Second := 59, [2].log_data[0].min := 1.0, [2].log_data[0].max := 1.0, [2].log_data[0].total := 300.0, [2].log_data[0].time := 300.0, [2].log_data[0].minminute := 30, [2].log_data[0].maxminute := 30, [2].log_data[0].valid := 1, [2].log_data[1].valid := 1, [2].log_data[2].valid := 1, [2].log_data[3].valid := 1, [2].log_data[4].valid := 1, [2].log_data[5].valid := 1, [2].log_data[6].valid := 1, [2].log_data[7].valid := 1, [2].log_data[8].valid := 1, [2].log_data[9].valid := 1, [2].log_data[10].valid := 1, [2].log_data[11].valid := 1, [2].log_data[12].valid := 1, [2].log_data[13].valid := 1, [2].log_data[14].valid := 1, [2].log_data[15].valid := 1, [2].log_data[16].valid := 1, [2].log_data[17].valid := 1, [2].log_data[18].valid := 1, [2].log_data[19].valid := 1, [2].time.Year := 2023, [2].time.Month := 1, [2].time.Day := 18, [2].time.Minute := 34, [2].time.Second := 59, [3].log_data[0].min := 1.0, [3].log_data[0].max := 1.0, [3].log_data[0].total := 300.0, [3].log_data[0].time := 300.0, [3].log_data[0].minminute := 35, [3].log_data[0].maxminute := 35, [3].log_data[0].valid := 1, [3].log_data[1].valid := 1, [3].log_data[2].valid := 1, [3].log_data[3].valid := 1, [3].log_data[4].valid := 1, [3].log_data[5].valid := 1, [3].log_data[6].valid := 1, [3].log_data[7].valid := 1, [3].log_data[8].valid := 1, [3].log_data[9].valid := 1, [3].log_data[10].valid := 1, [3].log_data[11].valid := 1, [3].log_data[12].valid := 1, [3].log_data[13].valid := 1, [3].log_data[14].valid := 1, [3].log_data[15].valid := 1, [3].log_data[16].valid := 1, [3].log_data[17].valid := 1, [3].log_data[18].valid := 1, [3].log_data[19].valid := 1, [3].time.Year := 2023,
        [3].time.Month := 1, [3].time.Day := 18, [3].time.Minute := 39, [3].time.Second := 59, [4].log_data[0].min := 1.0, [4].log_data[0].max := 1.0, [4].log_data[0].total := 300.0, [4].log_data[0].time := 300.0, [4].log_data[0].minminute := 40, [4].log_data[0].maxminute := 40, [4].log_data[0].valid := 1, [4].log_data[1].valid := 1, [4].log_data[2].valid := 1, [4].log_data[3].valid := 1, [4].log_data[4].valid := 1, [4].log_data[5].valid := 1, [4].log_data[6].valid := 1, [4].log_data[7].valid := 1, [4].log_data[8].valid := 1, [4].log_data[9].valid := 1, [4].log_data[10].valid := 1, [4].log_data[11].valid := 1, [4].log_data[12].valid := 1, [4].log_data[13].valid := 1, [4].log_data[14].valid := 1, [4].log_data[15].valid := 1, [4].log_data[16].valid := 1, [4].log_data[17].valid := 1, [4].log_data[18].valid := 1, [4].log_data[19].valid := 1, [4].time.Year := 2023, [4].time.Month := 1, [4].time.Day := 18, [4].time.Minute := 44, [4].time.Second := 59, [5].log_data[0].min := 1.0, [5].log_data[0].max := 1.0, [5].log_data[0].total := 300.0, [5].log_data[0].time := 300.0, [5].log_data[0].minminute := 45, [5].log_data[0].maxminute := 45, [5].log_data[0].valid := 1, [5].log_data[1].valid := 1, [5].log_data[2].valid := 1, [5].log_data[3].valid := 1, [5].log_data[4].valid := 1, [5].log_data[5].valid := 1, [5].log_data[6].valid := 1, [5].log_data[7].valid := 1, [5].log_data[8].valid := 1, [5].log_data[9].valid := 1, [5].log_data[10].valid := 1, [5].log_data[11].valid := 1, [5].log_data[12].valid := 1, [5].log_data[13].valid := 1, [5].log_data[14].valid := 1, [5].log_data[15].valid := 1, [5].log_data[16].valid := 1, [5].log_data[17].valid := 1, [5].log_data[18].valid := 1,
        [5].log_data[19].valid := 1, [5].time.Year := 2023, [5].time.Month := 1, [5].time.Day := 18, [5].time.Minute := 49, [5].time.Second := 59, [6].log_data[0].min := 1.0, [6].log_data[0].max := 1.0, [6].log_data[0].total := 300.0, [6].log_data[0].time := 300.0, [6].log_data[0].minminute := 50, [6].log_data[0].maxminute := 50, [6].log_data[0].valid := 1, [6].log_data[1].valid := 1, [6].log_data[2].valid := 1, [6].log_data[3].valid := 1, [6].log_data[4].valid := 1, [6].log_data[5].valid := 1, [6].log_data[6].valid := 1, [6].log_data[7].valid := 1, [6].log_data[8].valid := 1, [6].log_data[9].valid := 1, [6].log_data[10].valid := 1, [6].log_data[11].valid := 1, [6].log_data[12].valid := 1, [6].log_data[13].valid := 1, [6].log_data[14].valid := 1, [6].log_data[15].valid := 1, [6].log_data[16].valid := 1, [6].log_data[17].valid := 1, [6].log_data[18].valid := 1, [6].log_data[19].valid := 1, [6].time.Year := 2023, [6].time.Month := 1, [6].time.Day := 18, [6].time.Minute := 54, [6].time.Second := 59, [7].log_data[0].min := 1.0, [7].log_data[0].max := 1.0, [7].log_data[0].total := 300.0, [7].log_data[0].time := 300.0, [7].log_data[0].minminute := 55, [7].log_data[0].maxminute := 55, [7].log_data[0].valid := 1, [7].log_data[1].valid := 1, [7].log_data[2].valid := 1, [7].log_data[3].valid := 1, [7].log_data[4].valid := 1, [7].log_data[5].valid := 1, [7].log_data[6].valid := 1, [7].log_data[7].valid := 1, [7].log_data[8].valid := 1, [7].log_data[9].valid := 1, [7].log_data[10].valid := 1, [7].log_data[11].valid := 1, [7].log_data[12].valid := 1, [7].log_data[13].valid := 1, [7].log_data[14].valid := 1, [7].log_data[15].valid := 1, [7].log_data[16].valid := 1,
        [7].log_data[17].valid := 1, [7].log_data[18].valid := 1, [7].log_data[19].valid := 1, [7].time.Year := 2023, [7].time.Month := 1, [7].time.Day := 18, [7].time.Minute := 59, [7].time.Second := 59, [8].log_data[0].min := 1.0, [8].log_data[0].max := 1.0, [8].log_data[0].total := 300.0, [8].log_data[0].time := 300.0, [8].log_data[0].valid := 1, [8].log_data[1].valid := 1, [8].log_data[2].valid := 1, [8].log_data[3].valid := 1, [8].log_data[4].valid := 1, [8].log_data[5].valid := 1, [8].log_data[6].valid := 1, [8].log_data[7].valid := 1, [8].log_data[8].valid := 1, [8].log_data[9].valid := 1, [8].log_data[10].valid := 1, [8].log_data[11].valid := 1, [8].log_data[12].valid := 1, [8].log_data[13].valid := 1, [8].log_data[14].valid := 1, [8].log_data[15].valid := 1, [8].log_data[16].valid := 1, [8].log_data[17].valid := 1, [8].log_data[18].valid := 1, [8].log_data[19].valid := 1, [8].time.Year := 2023, [8].time.Month := 1, [8].time.Day := 18, [8].time.Hour := 1, [8].time.Minute := 4, [8].time.Second := 59, [9].log_data[0].min := 1.0, [9].log_data[0].max := 1.0, [9].log_data[0].total := 300.0, [9].log_data[0].time := 300.0, [9].log_data[0].minminute := 5, [9].log_data[0].maxminute := 5, [9].log_data[0].valid := 1, [9].log_data[1].valid := 1, [9].log_data[2].valid := 1, [9].log_data[3].valid := 1, [9].log_data[4].valid := 1, [9].log_data[5].valid := 1, [9].log_data[6].valid := 1, [9].log_data[7].valid := 1, [9].log_data[8].valid := 1, [9].log_data[9].valid := 1, [9].log_data[10].valid := 1, [9].log_data[11].valid := 1, [9].log_data[12].valid := 1, [9].log_data[13].valid := 1, [9].log_data[14].valid := 1, [9].log_data[15].valid := 1,
        [9].log_data[16].valid := 1, [9].log_data[17].valid := 1, [9].log_data[18].valid := 1, [9].log_data[19].valid := 1, [9].time.Year := 2023, [9].time.Month := 1, [9].time.Day := 18, [9].time.Hour := 1, [9].time.Minute := 9, [9].time.Second := 59, [10].log_data[0].min := 1.0, [10].log_data[0].max := 1.0, [10].log_data[0].total := 300.0, [10].log_data[0].time := 300.0, [10].log_data[0].minminute := 10, [10].log_data[0].maxminute := 10, [10].log_data[0].valid := 1, [10].log_data[1].valid := 1, [10].log_data[2].valid := 1, [10].log_data[3].valid := 1, [10].log_data[4].valid := 1, [10].log_data[5].valid := 1, [10].log_data[6].valid := 1, [10].log_data[7].valid := 1, [10].log_data[8].valid := 1, [10].log_data[9].valid := 1, [10].log_data[10].valid := 1, [10].log_data[11].valid := 1, [10].log_data[12].valid := 1, [10].log_data[13].valid := 1, [10].log_data[14].valid := 1, [10].log_data[15].valid := 1, [10].log_data[16].valid := 1, [10].log_data[17].valid := 1, [10].log_data[18].valid := 1, [10].log_data[19].valid := 1, [10].time.Year := 2023, [10].time.Month := 1, [10].time.Day := 18, [10].time.Hour := 1, [10].time.Minute := 14, [10].time.Second := 59, [11].log_data[0].min := 1.0, [11].log_data[0].max := 1.0, [11].log_data[0].total := 300.0, [11].log_data[0].time := 300.0, [11].log_data[0].minminute := 15, [11].log_data[0].maxminute := 15, [11].log_data[0].valid := 1, [11].log_data[1].valid := 1, [11].log_data[2].valid := 1, [11].log_data[3].valid := 1, [11].log_data[4].valid := 1, [11].log_data[5].valid := 1, [11].log_data[6].valid := 1, [11].log_data[7].valid := 1, [11].log_data[8].valid := 1, [11].log_data[9].valid := 1, [11].log_data[10].valid := 1, [11].log_data[11].valid := 1,
        [11].log_data[12].valid := 1, [11].log_data[13].valid := 1, [11].log_data[14].valid := 1, [11].log_data[15].valid := 1, [11].log_data[16].valid := 1, [11].log_data[17].valid := 1, [11].log_data[18].valid := 1, [11].log_data[19].valid := 1, [11].time.Year := 2023, [11].time.Month := 1, [11].time.Day := 18, [11].time.Hour := 1, [11].time.Minute := 19, [11].time.Second := 59, [12].log_data[0].min := 1.0, [12].log_data[0].max := 1.0, [12].log_data[0].total := 300.0, [12].log_data[0].time := 300.0, [12].log_data[0].minminute := 20, [12].log_data[0].maxminute := 20, [12].log_data[0].valid := 1, [12].log_data[1].valid := 1, [12].log_data[2].valid := 1, [12].log_data[3].valid := 1, [12].log_data[4].valid := 1, [12].log_data[5].valid := 1, [12].log_data[6].valid := 1, [12].log_data[7].valid := 1, [12].log_data[8].valid := 1, [12].log_data[9].valid := 1, [12].log_data[10].valid := 1, [12].log_data[11].valid := 1, [12].log_data[12].valid := 1, [12].log_data[13].valid := 1, [12].log_data[14].valid := 1, [12].log_data[15].valid := 1, [12].log_data[16].valid := 1, [12].log_data[17].valid := 1, [12].log_data[18].valid := 1, [12].log_data[19].valid := 1, [12].time.Year := 2023, [12].time.Month := 1, [12].time.Day := 18, [12].time.Hour := 1, [12].time.Minute := 24, [12].time.Second := 59, [13].log_data[0].min := 1.0, [13].log_data[0].max := 1.0, [13].log_data[0].total := 300.0, [13].log_data[0].time := 300.0, [13].log_data[0].minminute := 25, [13].log_data[0].maxminute := 25, [13].log_data[0].valid := 1, [13].log_data[1].valid := 1, [13].log_data[2].valid := 1, [13].log_data[3].valid := 1, [13].log_data[4].valid := 1, [13].log_data[5].valid := 1, [13].log_data[6].valid := 1, [13].log_data[7].valid := 1,
        [13].log_data[8].valid := 1, [13].log_data[9].valid := 1, [13].log_data[10].valid := 1, [13].log_data[11].valid := 1, [13].log_data[12].valid := 1, [13].log_data[13].valid := 1, [13].log_data[14].valid := 1, [13].log_data[15].valid := 1, [13].log_data[16].valid := 1, [13].log_data[17].valid := 1, [13].log_data[18].valid := 1, [13].log_data[19].valid := 1, [13].time.Year := 2023, [13].time.Month := 1, [13].time.Day := 18, [13].time.Hour := 1, [13].time.Minute := 29, [13].time.Second := 59, [14].log_data[0].min := 1.0, [14].log_data[0].max := 1.0, [14].log_data[0].total := 300.0, [14].log_data[0].time := 300.0, [14].log_data[0].minminute := 30, [14].log_data[0].maxminute := 30, [14].log_data[0].valid := 1, [14].log_data[1].valid := 1, [14].log_data[2].valid := 1, [14].log_data[3].valid := 1, [14].log_data[4].valid := 1, [14].log_data[5].valid := 1, [14].log_data[6].valid := 1, [14].log_data[7].valid := 1, [14].log_data[8].valid := 1, [14].log_data[9].valid := 1, [14].log_data[10].valid := 1, [14].log_data[11].valid := 1, [14].log_data[12].valid := 1, [14].log_data[13].valid := 1, [14].log_data[14].valid := 1, [14].log_data[15].valid := 1, [14].log_data[16].valid := 1, [14].log_data[17].valid := 1, [14].log_data[18].valid := 1, [14].log_data[19].valid := 1, [14].time.Year := 2023, [14].time.Month := 1, [14].time.Day := 18, [14].time.Hour := 1, [14].time.Minute := 34, [14].time.Second := 59, [15].log_data[0].min := 1.0, [15].log_data[0].max := 1.0, [15].log_data[0].total := 300.0, [15].log_data[0].time := 300.0, [15].log_data[0].minminute := 35, [15].log_data[0].maxminute := 35, [15].log_data[0].valid := 1, [15].log_data[1].valid := 1, [15].log_data[2].valid := 1, [15].log_data[3].valid := 1,
        [15].log_data[4].valid := 1, [15].log_data[5].valid := 1, [15].log_data[6].valid := 1, [15].log_data[7].valid := 1, [15].log_data[8].valid := 1, [15].log_data[9].valid := 1, [15].log_data[10].valid := 1, [15].log_data[11].valid := 1, [15].log_data[12].valid := 1, [15].log_data[13].valid := 1, [15].log_data[14].valid := 1, [15].log_data[15].valid := 1, [15].log_data[16].valid := 1, [15].log_data[17].valid := 1, [15].log_data[18].valid := 1, [15].log_data[19].valid := 1, [15].time.Year := 2023, [15].time.Month := 1, [15].time.Day := 18, [15].time.Hour := 1, [15].time.Minute := 39, [15].time.Second := 59, [16].log_data[0].min := 1.0, [16].log_data[0].max := 1.0, [16].log_data[0].total := 300.0, [16].log_data[0].time := 300.0, [16].log_data[0].minminute := 40, [16].log_data[0].maxminute := 40, [16].log_data[0].valid := 1, [16].log_data[1].valid := 1, [16].log_data[2].valid := 1, [16].log_data[3].valid := 1, [16].log_data[4].valid := 1, [16].log_data[5].valid := 1, [16].log_data[6].valid := 1, [16].log_data[7].valid := 1, [16].log_data[8].valid := 1, [16].log_data[9].valid := 1, [16].log_data[10].valid := 1, [16].log_data[11].valid := 1, [16].log_data[12].valid := 1, [16].log_data[13].valid := 1, [16].log_data[14].valid := 1, [16].log_data[15].valid := 1, [16].log_data[16].valid := 1, [16].log_data[17].valid := 1, [16].log_data[18].valid := 1, [16].log_data[19].valid := 1, [16].time.Year := 2023, [16].time.Month := 1, [16].time.Day := 18, [16].time.Hour := 1, [16].time.Minute := 44, [16].time.Second := 59, [17].log_data[0].min := 1.0, [17].log_data[0].max := 1.0, [17].log_data[0].total := 300.0, [17].log_data[0].time := 300.0, [17].log_data[0].minminute := 45, [17].log_data[0].maxminute := 45,
        [17].log_data[0].valid := 1, [17].log_data[1].valid := 1, [17].log_data[2].valid := 1, [17].log_data[3].valid := 1, [17].log_data[4].valid := 1, [17].log_data[5].valid := 1, [17].log_data[6].valid := 1, [17].log_data[7].valid := 1, [17].log_data[8].valid := 1, [17].log_data[9].valid := 1, [17].log_data[10].valid := 1, [17].log_data[11].valid := 1, [17].log_data[12].valid := 1, [17].log_data[13].valid := 1, [17].log_data[14].valid := 1, [17].log_data[15].valid := 1, [17].log_data[16].valid := 1, [17].log_data[17].valid := 1, [17].log_data[18].valid := 1, [17].log_data[19].valid := 1, [17].time.Year := 2023, [17].time.Month := 1, [17].time.Day := 18, [17].time.Hour := 1, [17].time.Minute := 49, [17].time.Second := 59, [18].log_data[0].min := 1.0, [18].log_data[0].max := 1.0, [18].log_data[0].total := 300.0, [18].log_data[0].time := 300.0, [18].log_data[0].minminute := 50, [18].log_data[0].maxminute := 50, [18].log_data[0].valid := 1, [18].log_data[1].valid := 1, [18].log_data[2].valid := 1, [18].log_data[3].valid := 1, [18].log_data[4].valid := 1, [18].log_data[5].valid := 1, [18].log_data[6].valid := 1, [18].log_data[7].valid := 1, [18].log_data[8].valid := 1, [18].log_data[9].valid := 1, [18].log_data[10].valid := 1, [18].log_data[11].valid := 1, [18].log_data[12].valid := 1, [18].log_data[13].valid := 1, [18].log_data[14].valid := 1, [18].log_data[15].valid := 1, [18].log_data[16].valid := 1, [18].log_data[17].valid := 1, [18].log_data[18].valid := 1, [18].log_data[19].valid := 1, [18].time.Year := 2023, [18].time.Month := 1, [18].time.Day := 18, [18].time.Hour := 1, [18].time.Minute := 54, [18].time.Second := 59, [19].log_data[0].min := 1.0, [19].log_data[0].max := 1.0,
        [19].log_data[0].total := 300.0, [19].log_data[0].time := 300.0, [19].log_data[0].minminute := 55, [19].log_data[0].maxminute := 55, [19].log_data[0].valid := 1, [19].log_data[1].valid := 1, [19].log_data[2].valid := 1, [19].log_data[3].valid := 1, [19].log_data[4].valid := 1, [19].log_data[5].valid := 1, [19].log_data[6].valid := 1, [19].log_data[7].valid := 1, [19].log_data[8].valid := 1, [19].log_data[9].valid := 1, [19].log_data[10].valid := 1, [19].log_data[11].valid := 1, [19].log_data[12].valid := 1, [19].log_data[13].valid := 1, [19].log_data[14].valid := 1, [19].log_data[15].valid := 1, [19].log_data[16].valid := 1, [19].log_data[17].valid := 1, [19].log_data[18].valid := 1, [19].log_data[19].valid := 1, [19].time.Year := 2023, [19].time.Month := 1, [19].time.Day := 18, [19].time.Hour := 1, [19].time.Minute := 59, [19].time.Second := 59, [20].log_data[0].min := 1.0, [20].log_data[0].max := 1.0, [20].log_data[0].total := 300.0, [20].log_data[0].time := 300.0, [20].log_data[0].valid := 1, [20].log_data[1].valid := 1, [20].log_data[2].valid := 1, [20].log_data[3].valid := 1, [20].log_data[4].valid := 1, [20].log_data[5].valid := 1, [20].log_data[6].valid := 1, [20].log_data[7].valid := 1, [20].log_data[8].valid := 1, [20].log_data[9].valid := 1, [20].log_data[10].valid := 1, [20].log_data[11].valid := 1, [20].log_data[12].valid := 1, [20].log_data[13].valid := 1, [20].log_data[14].valid := 1, [20].log_data[15].valid := 1, [20].log_data[16].valid := 1, [20].log_data[17].valid := 1, [20].log_data[18].valid := 1, [20].log_data[19].valid := 1, [20].time.Year := 2023, [20].time.Month := 1, [20].time.Day := 18, [20].time.Hour := 2, [20].time.Minute := 4, [20].time.Second := 59,
        [21].log_data[0].min := 1.0, [21].log_data[0].max := 1.0, [21].log_data[0].total := 300.0, [21].log_data[0].time := 300.0, [21].log_data[0].minminute := 5, [21].log_data[0].maxminute := 5, [21].log_data[0].valid := 1, [21].log_data[1].valid := 1, [21].log_data[2].valid := 1, [21].log_data[3].valid := 1, [21].log_data[4].valid := 1, [21].log_data[5].valid := 1, [21].log_data[6].valid := 1, [21].log_data[7].valid := 1, [21].log_data[8].valid := 1, [21].log_data[9].valid := 1, [21].log_data[10].valid := 1, [21].log_data[11].valid := 1, [21].log_data[12].valid := 1, [21].log_data[13].valid := 1, [21].log_data[14].valid := 1, [21].log_data[15].valid := 1, [21].log_data[16].valid := 1, [21].log_data[17].valid := 1, [21].log_data[18].valid := 1, [21].log_data[19].valid := 1, [21].time.Year := 2023, [21].time.Month := 1, [21].time.Day := 18, [21].time.Hour := 2, [21].time.Minute := 9, [21].time.Second := 59, [22].log_data[0].min := 1.0, [22].log_data[0].max := 1.0, [22].log_data[0].total := 300.0, [22].log_data[0].time := 300.0, [22].log_data[0].minminute := 10, [22].log_data[0].maxminute := 10, [22].log_data[0].valid := 1, [22].log_data[1].valid := 1, [22].log_data[2].valid := 1, [22].log_data[3].valid := 1, [22].log_data[4].valid := 1, [22].log_data[5].valid := 1, [22].log_data[6].valid := 1, [22].log_data[7].valid := 1, [22].log_data[8].valid := 1, [22].log_data[9].valid := 1, [22].log_data[10].valid := 1, [22].log_data[11].valid := 1, [22].log_data[12].valid := 1, [22].log_data[13].valid := 1, [22].log_data[14].valid := 1, [22].log_data[15].valid := 1, [22].log_data[16].valid := 1, [22].log_data[17].valid := 1, [22].log_data[18].valid := 1, [22].log_data[19].valid := 1, [22].time.Year := 2023, [22].time.Month := 1,
        [22].time.Day := 18, [22].time.Hour := 2, [22].time.Minute := 14, [22].time.Second := 59, [23].log_data[0].min := 1.0, [23].log_data[0].max := 1.0, [23].log_data[0].total := 300.0, [23].log_data[0].time := 300.0, [23].log_data[0].minminute := 15, [23].log_data[0].maxminute := 15, [23].log_data[0].valid := 1, [23].log_data[1].valid := 1, [23].log_data[2].valid := 1, [23].log_data[3].valid := 1, [23].log_data[4].valid := 1, [23].log_data[5].valid := 1, [23].log_data[6].valid := 1, [23].log_data[7].valid := 1, [23].log_data[8].valid := 1, [23].log_data[9].valid := 1, [23].log_data[10].valid := 1, [23].log_data[11].valid := 1, [23].log_data[12].valid := 1, [23].log_data[13].valid := 1, [23].log_data[14].valid := 1, [23].log_data[15].valid := 1, [23].log_data[16].valid := 1, [23].log_data[17].valid := 1, [23].log_data[18].valid := 1, [23].log_data[19].valid := 1, [23].time.Year := 2023, [23].time.Month := 1, [23].time.Day := 18, [23].time.Hour := 2, [23].time.Minute := 19, [23].time.Second := 59, [24].log_data[0].min := 1.0, [24].log_data[0].max := 1.0, [24].log_data[0].total := 300.0, [24].log_data[0].time := 300.0, [24].log_data[0].minminute := 20, [24].log_data[0].maxminute := 20, [24].log_data[0].valid := 1, [24].log_data[1].valid := 1, [24].log_data[2].valid := 1, [24].log_data[3].valid := 1, [24].log_data[4].valid := 1, [24].log_data[5].valid := 1, [24].log_data[6].valid := 1, [24].log_data[7].valid := 1, [24].log_data[8].valid := 1, [24].log_data[9].valid := 1, [24].log_data[10].valid := 1, [24].log_data[11].valid := 1, [24].log_data[12].valid := 1, [24].log_data[13].valid := 1, [24].log_data[14].valid := 1, [24].log_data[15].valid := 1, [24].log_data[16].valid := 1, [24].log_data[17].valid := 1,
        [24].log_data[18].valid := 1, [24].log_data[19].valid := 1, [24].time.Year := 2023, [24].time.Month := 1, [24].time.Day := 18, [24].time.Hour := 2, [24].time.Minute := 24, [24].time.Second := 59, [25].log_data[0].min := 1.0, [25].log_data[0].max := 1.0, [25].log_data[0].total := 300.0, [25].log_data[0].time := 300.0, [25].log_data[0].minminute := 25, [25].log_data[0].maxminute := 25, [25].log_data[0].valid := 1, [25].log_data[1].valid := 1, [25].log_data[2].valid := 1, [25].log_data[3].valid := 1, [25].log_data[4].valid := 1, [25].log_data[5].valid := 1, [25].log_data[6].valid := 1, [25].log_data[7].valid := 1, [25].log_data[8].valid := 1, [25].log_data[9].valid := 1, [25].log_data[10].valid := 1, [25].log_data[11].valid := 1, [25].log_data[12].valid := 1, [25].log_data[13].valid := 1, [25].log_data[14].valid := 1, [25].log_data[15].valid := 1, [25].log_data[16].valid := 1, [25].log_data[17].valid := 1, [25].log_data[18].valid := 1, [25].log_data[19].valid := 1, [25].time.Year := 2023, [25].time.Month := 1, [25].time.Day := 18, [25].time.Hour := 2, [25].time.Minute := 29, [25].time.Second := 59, [26].log_data[0].min := 1.0, [26].log_data[0].max := 1.0, [26].log_data[0].total := 300.0, [26].log_data[0].time := 300.0, [26].log_data[0].minminute := 30, [26].log_data[0].maxminute := 30, [26].log_data[0].valid := 1, [26].log_data[1].valid := 1, [26].log_data[2].valid := 1, [26].log_data[3].valid := 1, [26].log_data[4].valid := 1, [26].log_data[5].valid := 1, [26].log_data[6].valid := 1, [26].log_data[7].valid := 1, [26].log_data[8].valid := 1, [26].log_data[9].valid := 1, [26].log_data[10].valid := 1, [26].log_data[11].valid := 1, [26].log_data[12].valid := 1, [26].log_data[13].valid := 1,
        [26].log_data[14].valid := 1, [26].log_data[15].valid := 1, [26].log_data[16].valid := 1, [26].log_data[17].valid := 1, [26].log_data[18].valid := 1, [26].log_data[19].valid := 1, [26].time.Year := 2023, [26].time.Month := 1, [26].time.Day := 18, [26].time.Hour := 2, [26].time.Minute := 34, [26].time.Second := 59, [27].log_data[0].min := 1.0, [27].log_data[0].max := 1.0, [27].log_data[0].total := 300.0, [27].log_data[0].time := 300.0, [27].log_data[0].minminute := 35, [27].log_data[0].maxminute := 35, [27].log_data[0].valid := 1, [27].log_data[1].valid := 1, [27].log_data[2].valid := 1, [27].log_data[3].valid := 1, [27].log_data[4].valid := 1, [27].log_data[5].valid := 1, [27].log_data[6].valid := 1, [27].log_data[7].valid := 1, [27].log_data[8].valid := 1, [27].log_data[9].valid := 1, [27].log_data[10].valid := 1, [27].log_data[11].valid := 1, [27].log_data[12].valid := 1, [27].log_data[13].valid := 1, [27].log_data[14].valid := 1, [27].log_data[15].valid := 1, [27].log_data[16].valid := 1, [27].log_data[17].valid := 1, [27].log_data[18].valid := 1, [27].log_data[19].valid := 1, [27].time.Year := 2023, [27].time.Month := 1, [27].time.Day := 18, [27].time.Hour := 2, [27].time.Minute := 39, [27].time.Second := 59, [28].log_data[0].min := 1.0, [28].log_data[0].max := 1.0, [28].log_data[0].total := 300.0, [28].log_data[0].time := 300.0, [28].log_data[0].minminute := 40, [28].log_data[0].maxminute := 40, [28].log_data[0].valid := 1, [28].log_data[1].valid := 1, [28].log_data[2].valid := 1, [28].log_data[3].valid := 1, [28].log_data[4].valid := 1, [28].log_data[5].valid := 1, [28].log_data[6].valid := 1, [28].log_data[7].valid := 1, [28].log_data[8].valid := 1, [28].log_data[9].valid := 1,
        [28].log_data[10].valid := 1, [28].log_data[11].valid := 1, [28].log_data[12].valid := 1, [28].log_data[13].valid := 1, [28].log_data[14].valid := 1, [28].log_data[15].valid := 1, [28].log_data[16].valid := 1, [28].log_data[17].valid := 1, [28].log_data[18].valid := 1, [28].log_data[19].valid := 1, [28].time.Year := 2023, [28].time.Month := 1, [28].time.Day := 18, [28].time.Hour := 2, [28].time.Minute := 44, [28].time.Second := 59, [29].log_data[0].min := 1.0, [29].log_data[0].max := 1.0, [29].log_data[0].total := 300.0, [29].log_data[0].time := 300.0, [29].log_data[0].minminute := 45, [29].log_data[0].maxminute := 45, [29].log_data[0].valid := 1, [29].log_data[1].valid := 1, [29].log_data[2].valid := 1, [29].log_data[3].valid := 1, [29].log_data[4].valid := 1, [29].log_data[5].valid := 1, [29].log_data[6].valid := 1, [29].log_data[7].valid := 1, [29].log_data[8].valid := 1, [29].log_data[9].valid := 1, [29].log_data[10].valid := 1, [29].log_data[11].valid := 1, [29].log_data[12].valid := 1, [29].log_data[13].valid := 1, [29].log_data[14].valid := 1, [29].log_data[15].valid := 1, [29].log_data[16].valid := 1, [29].log_data[17].valid := 1, [29].log_data[18].valid := 1, [29].log_data[19].valid := 1, [29].time.Year := 2023, [29].time.Month := 1, [29].time.Day := 18, [29].time.Hour := 2, [29].time.Minute := 49, [29].time.Second := 59, [30].log_data[0].min := 1.0, [30].log_data[0].max := 1.0, [30].log_data[0].total := 300.0, [30].log_data[0].time := 300.0, [30].log_data[0].minminute := 50, [30].log_data[0].maxminute := 50, [30].log_data[0].valid := 1, [30].log_data[1].valid := 1, [30].log_data[2].valid := 1, [30].log_data[3].valid := 1, [30].log_data[4].valid := 1, [30].log_data[5].valid := 1,
        [30].log_data[6].valid := 1, [30].log_data[7].valid := 1, [30].log_data[8].valid := 1, [30].log_data[9].valid := 1, [30].log_data[10].valid := 1, [30].log_data[11].valid := 1, [30].log_data[12].valid := 1, [30].log_data[13].valid := 1, [30].log_data[14].valid := 1, [30].log_data[15].valid := 1, [30].log_data[16].valid := 1, [30].log_data[17].valid := 1, [30].log_data[18].valid := 1, [30].log_data[19].valid := 1, [30].time.Year := 2023, [30].time.Month := 1, [30].time.Day := 18, [30].time.Hour := 2, [30].time.Minute := 54, [30].time.Second := 59, [31].log_data[0].min := 1.0, [31].log_data[0].max := 1.0, [31].log_data[0].total := 300.0, [31].log_data[0].time := 300.0, [31].log_data[0].minminute := 55, [31].log_data[0].maxminute := 55, [31].log_data[0].valid := 1, [31].log_data[1].valid := 1, [31].log_data[2].valid := 1, [31].log_data[3].valid := 1, [31].log_data[4].valid := 1, [31].log_data[5].valid := 1, [31].log_data[6].valid := 1, [31].log_data[7].valid := 1, [31].log_data[8].valid := 1, [31].log_data[9].valid := 1, [31].log_data[10].valid := 1, [31].log_data[11].valid := 1, [31].log_data[12].valid := 1, [31].log_data[13].valid := 1, [31].log_data[14].valid := 1, [31].log_data[15].valid := 1, [31].log_data[16].valid := 1, [31].log_data[17].valid := 1, [31].log_data[18].valid := 1, [31].log_data[19].valid := 1, [31].time.Year := 2023, [31].time.Month := 1, [31].time.Day := 18, [31].time.Hour := 2, [31].time.Minute := 59, [31].time.Second := 59, [32].log_data[0].min := 1.0, [32].log_data[0].max := 1.0, [32].log_data[0].total := 300.0, [32].log_data[0].time := 300.0, [32].log_data[0].valid := 1, [32].log_data[1].valid := 1, [32].log_data[2].valid := 1, [32].log_data[3].valid := 1,
        [32].log_data[4].valid := 1, [32].log_data[5].valid := 1, [32].log_data[6].valid := 1, [32].log_data[7].valid := 1, [32].log_data[8].valid := 1, [32].log_data[9].valid := 1, [32].log_data[10].valid := 1, [32].log_data[11].valid := 1, [32].log_data[12].valid := 1, [32].log_data[13].valid := 1, [32].log_data[14].valid := 1, [32].log_data[15].valid := 1, [32].log_data[16].valid := 1, [32].log_data[17].valid := 1, [32].log_data[18].valid := 1, [32].log_data[19].valid := 1, [32].time.Year := 2023, [32].time.Month := 1, [32].time.Day := 18, [32].time.Hour := 3, [32].time.Minute := 4, [32].time.Second := 59, [33].log_data[0].min := 1.0, [33].log_data[0].max := 1.0, [33].log_data[0].total := 300.0, [33].log_data[0].time := 300.0, [33].log_data[0].minminute := 5, [33].log_data[0].maxminute := 5, [33].log_data[0].valid := 1, [33].log_data[1].valid := 1, [33].log_data[2].valid := 1, [33].log_data[3].valid := 1, [33].log_data[4].valid := 1, [33].log_data[5].valid := 1, [33].log_data[6].valid := 1, [33].log_data[7].valid := 1, [33].log_data[8].valid := 1, [33].log_data[9].valid := 1, [33].log_data[10].valid := 1, [33].log_data[11].valid := 1, [33].log_data[12].valid := 1, [33].log_data[13].valid := 1, [33].log_data[14].valid := 1, [33].log_data[15].valid := 1, [33].log_data[16].valid := 1, [33].log_data[17].valid := 1, [33].log_data[18].valid := 1, [33].log_data[19].valid := 1, [33].time.Year := 2023, [33].time.Month := 1, [33].time.Day := 18, [33].time.Hour := 3, [33].time.Minute := 9, [33].time.Second := 59, [34].log_data[0].min := 1.0, [34].log_data[0].max := 1.0, [34].log_data[0].total := 300.0, [34].log_data[0].time := 300.0, [34].log_data[0].minminute := 10, [34].log_data[0].maxminute := 10,
        [34].log_data[0].valid := 1, [34].log_data[1].valid := 1, [34].log_data[2].valid := 1, [34].log_data[3].valid := 1, [34].log_data[4].valid := 1, [34].log_data[5].valid := 1, [34].log_data[6].valid := 1, [34].log_data[7].valid := 1, [34].log_data[8].valid := 1, [34].log_data[9].valid := 1, [34].log_data[10].valid := 1, [34].log_data[11].valid := 1, [34].log_data[12].valid := 1, [34].log_data[13].valid := 1, [34].log_data[14].valid := 1, [34].log_data[15].valid := 1, [34].log_data[16].valid := 1, [34].log_data[17].valid := 1, [34].log_data[18].valid := 1, [34].log_data[19].valid := 1, [34].time.Year := 2023, [34].time.Month := 1, [34].time.Day := 18, [34].time.Hour := 3, [34].time.Minute := 14, [34].time.Second := 59, [35].log_data[0].min := 1.0, [35].log_data[0].max := 1.0, [35].log_data[0].total := 300.0, [35].log_data[0].time := 300.0, [35].log_data[0].minminute := 15, [35].log_data[0].maxminute := 15, [35].log_data[0].valid := 1, [35].log_data[1].valid := 1, [35].log_data[2].valid := 1, [35].log_data[3].valid := 1, [35].log_data[4].valid := 1, [35].log_data[5].valid := 1, [35].log_data[6].valid := 1, [35].log_data[7].valid := 1, [35].log_data[8].valid := 1, [35].log_data[9].valid := 1, [35].log_data[10].valid := 1, [35].log_data[11].valid := 1, [35].log_data[12].valid := 1, [35].log_data[13].valid := 1, [35].log_data[14].valid := 1, [35].log_data[15].valid := 1, [35].log_data[16].valid := 1, [35].log_data[17].valid := 1, [35].log_data[18].valid := 1, [35].log_data[19].valid := 1, [35].time.Year := 2023, [35].time.Month := 1, [35].time.Day := 18, [35].time.Hour := 3, [35].time.Minute := 19, [35].time.Second := 59, [36].log_data[0].min := 1.0, [36].log_data[0].max := 1.0,
        [36].log_data[0].total := 300.0, [36].log_data[0].time := 300.0, [36].log_data[0].minminute := 20, [36].log_data[0].maxminute := 20, [36].log_data[0].valid := 1, [36].log_data[1].valid := 1, [36].log_data[2].valid := 1, [36].log_data[3].valid := 1, [36].log_data[4].valid := 1, [36].log_data[5].valid := 1, [36].log_data[6].valid := 1, [36].log_data[7].valid := 1, [36].log_data[8].valid := 1, [36].log_data[9].valid := 1, [36].log_data[10].valid := 1, [36].log_data[11].valid := 1, [36].log_data[12].valid := 1, [36].log_data[13].valid := 1, [36].log_data[14].valid := 1, [36].log_data[15].valid := 1, [36].log_data[16].valid := 1, [36].log_data[17].valid := 1, [36].log_data[18].valid := 1, [36].log_data[19].valid := 1, [36].time.Year := 2023, [36].time.Month := 1, [36].time.Day := 18, [36].time.Hour := 3, [36].time.Minute := 24, [36].time.Second := 59, [37].log_data[0].min := 1.0, [37].log_data[0].max := 1.0, [37].log_data[0].total := 300.0, [37].log_data[0].time := 300.0, [37].log_data[0].minminute := 25, [37].log_data[0].maxminute := 25, [37].log_data[0].valid := 1, [37].log_data[1].valid := 1, [37].log_data[2].valid := 1, [37].log_data[3].valid := 1, [37].log_data[4].valid := 1, [37].log_data[5].valid := 1, [37].log_data[6].valid := 1, [37].log_data[7].valid := 1, [37].log_data[8].valid := 1, [37].log_data[9].valid := 1, [37].log_data[10].valid := 1, [37].log_data[11].valid := 1, [37].log_data[12].valid := 1, [37].log_data[13].valid := 1, [37].log_data[14].valid := 1, [37].log_data[15].valid := 1, [37].log_data[16].valid := 1, [37].log_data[17].valid := 1, [37].log_data[18].valid := 1, [37].log_data[19].valid := 1, [37].time.Year := 2023, [37].time.Month := 1, [37].time.Day := 18, [37].time.Hour := 3,
        [37].time.Minute := 29, [37].time.Second := 59, [38].log_data[0].min := 1.0, [38].log_data[0].max := 1.0, [38].log_data[0].total := 300.0, [38].log_data[0].time := 300.0, [38].log_data[0].minminute := 30, [38].log_data[0].maxminute := 30, [38].log_data[0].valid := 1, [38].log_data[1].valid := 1, [38].log_data[2].valid := 1, [38].log_data[3].valid := 1, [38].log_data[4].valid := 1, [38].log_data[5].valid := 1, [38].log_data[6].valid := 1, [38].log_data[7].valid := 1, [38].log_data[8].valid := 1, [38].log_data[9].valid := 1, [38].log_data[10].valid := 1, [38].log_data[11].valid := 1, [38].log_data[12].valid := 1, [38].log_data[13].valid := 1, [38].log_data[14].valid := 1, [38].log_data[15].valid := 1, [38].log_data[16].valid := 1, [38].log_data[17].valid := 1, [38].log_data[18].valid := 1, [38].log_data[19].valid := 1, [38].time.Year := 2023, [38].time.Month := 1, [38].time.Day := 18, [38].time.Hour := 3, [38].time.Minute := 34, [38].time.Second := 59, [39].log_data[0].min := 1.0, [39].log_data[0].max := 1.0, [39].log_data[0].total := 300.0, [39].log_data[0].time := 300.0, [39].log_data[0].minminute := 35, [39].log_data[0].maxminute := 35, [39].log_data[0].valid := 1, [39].log_data[1].valid := 1, [39].log_data[2].valid := 1, [39].log_data[3].valid := 1, [39].log_data[4].valid := 1, [39].log_data[5].valid := 1, [39].log_data[6].valid := 1, [39].log_data[7].valid := 1, [39].log_data[8].valid := 1, [39].log_data[9].valid := 1, [39].log_data[10].valid := 1, [39].log_data[11].valid := 1, [39].log_data[12].valid := 1, [39].log_data[13].valid := 1, [39].log_data[14].valid := 1, [39].log_data[15].valid := 1, [39].log_data[16].valid := 1, [39].log_data[17].valid := 1, [39].log_data[18].valid := 1, [39].log_data[19].valid := 1,
        [39].time.Year := 2023, [39].time.Month := 1, [39].time.Day := 18, [39].time.Hour := 3, [39].time.Minute := 39, [39].time.Second := 59, [40].log_data[0].min := 1.0, [40].log_data[0].max := 1.0, [40].log_data[0].total := 300.0, [40].log_data[0].time := 300.0, [40].log_data[0].minminute := 40, [40].log_data[0].maxminute := 40, [40].log_data[0].valid := 1, [40].log_data[1].valid := 1, [40].log_data[2].valid := 1, [40].log_data[3].valid := 1, [40].log_data[4].valid := 1, [40].log_data[5].valid := 1, [40].log_data[6].valid := 1, [40].log_data[7].valid := 1, [40].log_data[8].valid := 1, [40].log_data[9].valid := 1, [40].log_data[10].valid := 1, [40].log_data[11].valid := 1, [40].log_data[12].valid := 1, [40].log_data[13].valid := 1, [40].log_data[14].valid := 1, [40].log_data[15].valid := 1, [40].log_data[16].valid := 1, [40].log_data[17].valid := 1, [40].log_data[18].valid := 1, [40].log_data[19].valid := 1, [40].time.Year := 2023, [40].time.Month := 1, [40].time.Day := 18, [40].time.Hour := 3, [40].time.Minute := 44, [40].time.Second := 59, [41].log_data[0].min := 1.0, [41].log_data[0].max := 1.0, [41].log_data[0].total := 300.0, [41].log_data[0].time := 300.0, [41].log_data[0].minminute := 45, [41].log_data[0].maxminute := 45, [41].log_data[0].valid := 1, [41].log_data[1].valid := 1, [41].log_data[2].valid := 1, [41].log_data[3].valid := 1, [41].log_data[4].valid := 1, [41].log_data[5].valid := 1, [41].log_data[6].valid := 1, [41].log_data[7].valid := 1, [41].log_data[8].valid := 1, [41].log_data[9].valid := 1, [41].log_data[10].valid := 1, [41].log_data[11].valid := 1, [41].log_data[12].valid := 1, [41].log_data[13].valid := 1, [41].log_data[14].valid := 1, [41].log_data[15].valid := 1,
